   1:  PR[GP1:91,1] = PR[GP1:90,1] + 27.074;
   1:  PR[GP1:91,2] = PR[GP1:90,2] + -9.305;
   1:L PR[91] R[100]mm/sec CNT100;
   1:  PR[GP1:91,1] = PR[GP1:90,1] + 28.052;
   1:  PR[GP1:91,2] = PR[GP1:90,2] + -6.402;
   1:L PR[91] R[100]mm/sec CNT100;
   1:  PR[GP1:91,1] = PR[GP1:90,1] + 28.426;
   1:  PR[GP1:91,2] = PR[GP1:90,2] + -3.528;
   1:L PR[91] R[100]mm/sec CNT100;
   1:  PR[GP1:91,1] = PR[GP1:90,1] + 28.781;
   1:  PR[GP1:91,2] = PR[GP1:90,2] + -0.326;
   1:L PR[91] R[100]mm/sec CNT100;
   1:  PR[GP1:91,1] = PR[GP1:90,1] + 28.412;
   1:  PR[GP1:91,2] = PR[GP1:90,2] + 2.511;
   1:L PR[91] R[100]mm/sec CNT100;
   1:  PR[GP1:91,1] = PR[GP1:90,1] + 28.089;
   1:  PR[GP1:91,2] = PR[GP1:90,2] + 5.607;
   1:L PR[91] R[100]mm/sec CNT100;
   1:  PR[GP1:91,1] = PR[GP1:90,1] + 27.206;
   1:  PR[GP1:91,2] = PR[GP1:90,2] + 8.384;
   1:L PR[91] R[100]mm/sec CNT100;
   1:  PR[GP1:91,1] = PR[GP1:90,1] + 26.117;
   1:  PR[GP1:91,2] = PR[GP1:90,2] + 11.033;
   1:L PR[91] R[100]mm/sec CNT100;
   1:  PR[GP1:91,1] = PR[GP1:90,1] + 24.650;
   1:  PR[GP1:91,2] = PR[GP1:90,2] + 13.658;
   1:L PR[91] R[100]mm/sec CNT100;
   1:  PR[GP1:91,1] = PR[GP1:90,1] + 22.947;
   1:  PR[GP1:91,2] = PR[GP1:90,2] + 15.921;
   1:L PR[91] R[100]mm/sec CNT100;
   1:  PR[GP1:91,1] = PR[GP1:90,1] + 20.753;
   1:  PR[GP1:91,2] = PR[GP1:90,2] + 18.419;
   1:L PR[91] R[100]mm/sec CNT100;
   1:  PR[GP1:91,1] = PR[GP1:90,1] + 18.590;
   1:  PR[GP1:91,2] = PR[GP1:90,2] + 20.133;
   1:L PR[91] R[100]mm/sec CNT100;
   1:  PR[GP1:91,1] = PR[GP1:90,1] + 15.465;
   1:  PR[GP1:91,2] = PR[GP1:90,2] + 22.345;
   1:L PR[91] R[100]mm/sec CNT100;
   1:  PR[GP1:91,1] = PR[GP1:90,1] + 13.026;
   1:  PR[GP1:91,2] = PR[GP1:90,2] + 23.427;
   1:L PR[91] R[100]mm/sec CNT100;
   1:  PR[GP1:91,1] = PR[GP1:90,1] + 9.359;
   1:  PR[GP1:91,2] = PR[GP1:90,2] + 24.848;
   1:L PR[91] R[100]mm/sec CNT100;
   1:  PR[GP1:91,1] = PR[GP1:90,1] + 6.820;
   1:  PR[GP1:91,2] = PR[GP1:90,2] + 25.271;
   1:L PR[91] R[100]mm/sec CNT100;
   1:  PR[GP1:91,1] = PR[GP1:90,1] + 2.805;
   1:  PR[GP1:91,2] = PR[GP1:90,2] + 25.769;
   1:L PR[91] R[100]mm/sec CNT100;
   1:  PR[GP1:91,1] = PR[GP1:90,1] + 0.266;
   1:  PR[GP1:91,2] = PR[GP1:90,2] + 25.578;
   1:L PR[91] R[100]mm/sec CNT100;
   1:  PR[91] = PR[90];
   1:  PR[GP1:91,1] = PR[GP1:90,1] + -0.092;
   1:  PR[GP1:91,2] = PR[GP1:90,2] + 25.736;
   1:  PR[GP1:91,3] = PR[GP1:90,3] + 68.625;
   1:L PR[91] R[100]mm/sec CNT100;
   1:  PR[GP1:91,1] = PR[GP1:90,1] + -2.390;
   1:  PR[GP1:91,2] = PR[GP1:90,2] + 25.906;
   1:L PR[91] R[100]mm/sec CNT100;
   1:  PR[GP1:91,1] = PR[GP1:90,1] + -6.675;
   1:  PR[GP1:91,2] = PR[GP1:90,2] + 25.375;
   1:L PR[91] R[100]mm/sec CNT100;
   1:  PR[GP1:91,1] = PR[GP1:90,1] + -8.961;
   1:  PR[GP1:91,2] = PR[GP1:90,2] + 24.994;
   1:L PR[91] R[100]mm/sec CNT100;
   1:  PR[GP1:91,1] = PR[GP1:90,1] + -12.889;
   1:  PR[GP1:91,2] = PR[GP1:90,2] + 23.472;
   1:L PR[91] R[100]mm/sec CNT100;
   1:  PR[GP1:91,1] = PR[GP1:90,1] + -15.085;
   1:  PR[GP1:91,2] = PR[GP1:90,2] + 22.498;
   1:L PR[91] R[100]mm/sec CNT100;
   1:  PR[GP1:91,1] = PR[GP1:90,1] + -18.448;
   1:  PR[GP1:91,2] = PR[GP1:90,2] + 20.117;
   1:L PR[91] R[100]mm/sec CNT100;
   1:  PR[GP1:91,1] = PR[GP1:90,1] + -20.400;
   1:  PR[GP1:91,2] = PR[GP1:90,2] + 18.570;
   1:L PR[91] R[100]mm/sec CNT100;
   1:  PR[GP1:91,1] = PR[GP1:90,1] + -22.619;
   1:  PR[GP1:91,2] = PR[GP1:90,2] + 16.084;
   1:L PR[91] R[100]mm/sec CNT100;
   1:  PR[GP1:91,1] = PR[GP1:90,1] + -24.160;
   1:  PR[GP1:91,2] = PR[GP1:90,2] + 14.037;
   1:L PR[91] R[100]mm/sec CNT100;
   1:  PR[GP1:91,1] = PR[GP1:90,1] + -25.748;
   1:  PR[GP1:91,2] = PR[GP1:90,2] + 11.314;
   1:L PR[91] R[100]mm/sec CNT100;
   1:  PR[GP1:91,1] = PR[GP1:90,1] + -26.729;
   1:  PR[GP1:91,2] = PR[GP1:90,2] + 8.924;
   1:L PR[91] R[100]mm/sec CNT100;
   1:  PR[GP1:91,1] = PR[GP1:90,1] + -27.794;
   1:  PR[GP1:91,2] = PR[GP1:90,2] + 5.767;
   1:L PR[91] R[100]mm/sec CNT100;
   1:  PR[GP1:91,1] = PR[GP1:90,1] + -28.130;
   1:  PR[GP1:91,2] = PR[GP1:90,2] + 3.188;
   1:L PR[91] R[100]mm/sec CNT100;
   1:  PR[GP1:91,1] = PR[GP1:90,1] + -28.516;
   1:  PR[GP1:91,2] = PR[GP1:90,2] + -0.298;
   1:L PR[91] R[100]mm/sec CNT100;
   1:  PR[GP1:91,1] = PR[GP1:90,1] + -28.184;
   1:  PR[GP1:91,2] = PR[GP1:90,2] + -2.847;
   1:L PR[91] R[100]mm/sec CNT100;
   1:  PR[GP1:91,1] = PR[GP1:90,1] + -27.833;
   1:  PR[GP1:91,2] = PR[GP1:90,2] + -6.208;
   1:L PR[91] R[100]mm/sec CNT100;
   1:  PR[GP1:91,1] = PR[GP1:90,1] + -26.872;
   1:  PR[GP1:91,2] = PR[GP1:90,2] + -9.231;
   1:L PR[91] R[100]mm/sec CNT100;
   1:  PR[GP1:91,1] = PR[GP1:90,1] + -25.890;
   1:  PR[GP1:91,2] = PR[GP1:90,2] + -11.618;
   1:L PR[91] R[100]mm/sec CNT100;
   1:  PR[GP1:91,1] = PR[GP1:90,1] + -24.299;
   1:  PR[GP1:91,2] = PR[GP1:90,2] + -14.466;
   1:L PR[91] R[100]mm/sec CNT100;
   1:  PR[GP1:91,1] = PR[GP1:90,1] + -22.763;
   1:  PR[GP1:91,2] = PR[GP1:90,2] + -16.503;
   1:L PR[91] R[100]mm/sec CNT100;
   1:  PR[GP1:91,1] = PR[GP1:90,1] + -20.390;
   1:  PR[GP1:91,2] = PR[GP1:90,2] + -19.204;
   1:L PR[91] R[100]mm/sec CNT100;
   1:  PR[GP1:91,1] = PR[GP1:90,1] + -16.718;
   1:  PR[GP1:91,2] = PR[GP1:90,2] + -22.122;
   1:L PR[91] R[100]mm/sec CNT100;
   1:  PR[GP1:91,1] = PR[GP1:90,1] + -14.983;
   1:  PR[GP1:91,2] = PR[GP1:90,2] + -23.178;
   1:L PR[91] R[100]mm/sec CNT100;
   1:  PR[GP1:91,1] = PR[GP1:90,1] + -12.771;
   1:  PR[GP1:91,2] = PR[GP1:90,2] + -24.157;
   1:L PR[91] R[100]mm/sec CNT100;
   1:  PR[GP1:91,1] = PR[GP1:90,1] + -8.827;
   1:  PR[GP1:91,2] = PR[GP1:90,2] + -25.648;
   1:L PR[91] R[100]mm/sec CNT100;
   1:  PR[GP1:91,1] = PR[GP1:90,1] + -6.599;
   1:  PR[GP1:91,2] = PR[GP1:90,2] + -26.016;
   1:L PR[91] R[100]mm/sec CNT100;
   1:  PR[GP1:91,1] = PR[GP1:90,1] + -2.291;
   1:  PR[GP1:91,2] = PR[GP1:90,2] + -26.524;
   1:L PR[91] R[100]mm/sec CNT100;
   1:  PR[GP1:91,1] = PR[GP1:90,1] + -0.100;
   1:  PR[GP1:91,2] = PR[GP1:90,2] + -26.354;
   1:L PR[91] R[100]mm/sec CNT100;
   1:  PR[GP1:91,1] = PR[GP1:90,1] + 0.256;
   1:L PR[91] R[100]mm/sec CNT100;
   1:  PR[GP1:91,1] = PR[GP1:90,1] + 2.490;
   1:  PR[GP1:91,2] = PR[GP1:90,2] + -26.527;
   1:L PR[91] R[100]mm/sec CNT100;
   1:  PR[GP1:91,1] = PR[GP1:90,1] + 4.700;
   1:  PR[GP1:91,2] = PR[GP1:90,2] + -26.395;
   1:L PR[91] R[100]mm/sec CNT100;
   1:  PR[GP1:91,1] = PR[GP1:90,1] + 7.039;
   1:  PR[GP1:91,2] = PR[GP1:90,2] + -26.007;
   1:L PR[91] R[100]mm/sec CNT100;
   1:  PR[GP1:91,1] = PR[GP1:90,1] + 9.138;
   1:  PR[GP1:91,2] = PR[GP1:90,2] + -25.611;
   1:L PR[91] R[100]mm/sec CNT100;
   1:  PR[GP1:91,1] = PR[GP1:90,1] + 13.058;
   1:  PR[GP1:91,2] = PR[GP1:90,2] + -24.087;
   1:L PR[91] R[100]mm/sec CNT100;
   1:  PR[GP1:91,1] = PR[GP1:90,1] + 15.230;
   1:  PR[GP1:91,2] = PR[GP1:90,2] + -23.127;
   1:L PR[91] R[100]mm/sec CNT100;
   1:  PR[GP1:91,1] = PR[GP1:90,1] + 18.598;
   1:  PR[GP1:91,2] = PR[GP1:90,2] + -20.745;
   1:L PR[91] R[100]mm/sec CNT100;
   1:  PR[GP1:91,1] = PR[GP1:90,1] + 20.553;
   1:  PR[GP1:91,2] = PR[GP1:90,2] + -19.198;
   1:L PR[91] R[100]mm/sec CNT100;
   1:  PR[GP1:91,1] = PR[GP1:90,1] + 22.771;
   1:  PR[GP1:91,2] = PR[GP1:90,2] + -16.712;
   1:L PR[91] R[100]mm/sec CNT100;
   1:  PR[GP1:91,1] = PR[GP1:90,1] + 24.315;
   1:  PR[GP1:91,2] = PR[GP1:90,2] + -14.663;
   1:L PR[91] R[100]mm/sec CNT100;
   1:  PR[GP1:91,1] = PR[GP1:90,1] + 25.903;
   1:  PR[GP1:91,2] = PR[GP1:90,2] + -11.940;
   1:L PR[91] R[100]mm/sec CNT100;
   1:  PR[GP1:91,1] = PR[GP1:90,1] + 26.886;
   1:  PR[GP1:91,2] = PR[GP1:90,2] + -9.552;
   1:L PR[91] R[100]mm/sec CNT100;
   1:  PR[GP1:91,1] = PR[GP1:90,1] + 27.950;
   1:  PR[GP1:91,2] = PR[GP1:90,2] + -6.395;
   1:L PR[91] R[100]mm/sec CNT100;
   1:  PR[GP1:91,1] = PR[GP1:90,1] + 28.287;
   1:  PR[GP1:91,2] = PR[GP1:90,2] + -3.812;
   1:L PR[91] R[100]mm/sec CNT100;
   1:  PR[GP1:91,1] = PR[GP1:90,1] + 28.673;
   1:  PR[GP1:91,2] = PR[GP1:90,2] + -0.326;
   1:L PR[91] R[100]mm/sec CNT100;
   1:  PR[GP1:91,1] = PR[GP1:90,1] + 28.341;
   1:  PR[GP1:91,2] = PR[GP1:90,2] + 2.223;
   1:L PR[91] R[100]mm/sec CNT100;
   1:  PR[GP1:91,1] = PR[GP1:90,1] + 27.991;
   1:  PR[GP1:91,2] = PR[GP1:90,2] + 5.583;
   1:L PR[91] R[100]mm/sec CNT100;
   1:  PR[GP1:91,1] = PR[GP1:90,1] + 27.030;
   1:  PR[GP1:91,2] = PR[GP1:90,2] + 8.605;
   1:L PR[91] R[100]mm/sec CNT100;
   1:  PR[GP1:91,1] = PR[GP1:90,1] + 26.050;
   1:  PR[GP1:91,2] = PR[GP1:90,2] + 10.988;
   1:L PR[91] R[100]mm/sec CNT100;
   1:  PR[GP1:91,1] = PR[GP1:90,1] + 24.458;
   1:  PR[GP1:91,2] = PR[GP1:90,2] + 13.836;
   1:L PR[91] R[100]mm/sec CNT100;
   1:  PR[GP1:91,1] = PR[GP1:90,1] + 22.926;
   1:  PR[GP1:91,2] = PR[GP1:90,2] + 15.873;
   1:L PR[91] R[100]mm/sec CNT100;
   1:  PR[GP1:91,1] = PR[GP1:90,1] + 20.554;
   1:  PR[GP1:91,2] = PR[GP1:90,2] + 18.573;
   1:L PR[91] R[100]mm/sec CNT100;
   1:  PR[GP1:91,1] = PR[GP1:90,1] + 18.605;
   1:  PR[GP1:91,2] = PR[GP1:90,2] + 20.117;
   1:L PR[91] R[100]mm/sec CNT100;
   1:  PR[GP1:91,1] = PR[GP1:90,1] + 15.243;
   1:  PR[GP1:91,2] = PR[GP1:90,2] + 22.498;
   1:L PR[91] R[100]mm/sec CNT100;
   1:  PR[GP1:91,1] = PR[GP1:90,1] + 13.047;
   1:  PR[GP1:91,2] = PR[GP1:90,2] + 23.472;
   1:L PR[91] R[100]mm/sec CNT100;
   1:  PR[GP1:91,1] = PR[GP1:90,1] + 9.117;
   1:  PR[GP1:91,2] = PR[GP1:90,2] + 24.994;
   1:L PR[91] R[100]mm/sec CNT100;
   1:  PR[GP1:91,1] = PR[GP1:90,1] + 6.832;
   1:  PR[GP1:91,2] = PR[GP1:90,2] + 25.375;
   1:L PR[91] R[100]mm/sec CNT100;
   1:  PR[GP1:91,1] = PR[GP1:90,1] + 2.546;
   1:  PR[GP1:91,2] = PR[GP1:90,2] + 25.906;
   1:L PR[91] R[100]mm/sec CNT100;
   1:  PR[GP1:91,1] = PR[GP1:90,1] + 0.252;
   1:  PR[GP1:91,2] = PR[GP1:90,2] + 25.736;
   1:L PR[91] R[100]mm/sec CNT100;
   1:  PR[91] = PR[90];
   1:  PR[GP1:91,1] = PR[GP1:90,1] + -0.083;
   1:  PR[GP1:91,2] = PR[GP1:90,2] + 25.892;
   1:  PR[GP1:91,3] = PR[GP1:90,3] + 69.235;
   1:L PR[91] R[100]mm/sec CNT100;
   1:  PR[GP1:91,1] = PR[GP1:90,1] + -2.132;
   1:  PR[GP1:91,2] = PR[GP1:90,2] + 26.044;
   1:L PR[91] R[100]mm/sec CNT100;
   1:  PR[GP1:91,1] = PR[GP1:90,1] + -6.687;
   1:  PR[GP1:91,2] = PR[GP1:90,2] + 25.479;
   1:L PR[91] R[100]mm/sec CNT100;
   1:  PR[GP1:91,1] = PR[GP1:90,1] + -8.719;
   1:  PR[GP1:91,2] = PR[GP1:90,2] + 25.141;
   1:L PR[91] R[100]mm/sec CNT100;
   1:  PR[GP1:91,1] = PR[GP1:90,1] + -12.910;
   1:  PR[GP1:91,2] = PR[GP1:90,2] + 23.517;
   1:L PR[91] R[100]mm/sec CNT100;
   1:  PR[GP1:91,1] = PR[GP1:90,1] + -14.863;
   1:  PR[GP1:91,2] = PR[GP1:90,2] + 22.650;
   1:L PR[91] R[100]mm/sec CNT100;
   1:  PR[GP1:91,1] = PR[GP1:90,1] + -18.463;
   1:  PR[GP1:91,2] = PR[GP1:90,2] + 20.101;
   1:L PR[91] R[100]mm/sec CNT100;
   1:  PR[GP1:91,1] = PR[GP1:90,1] + -20.201;
   1:  PR[GP1:91,2] = PR[GP1:90,2] + 18.724;
   1:L PR[91] R[100]mm/sec CNT100;
   1:  PR[GP1:91,1] = PR[GP1:90,1] + -22.586;
   1:  PR[GP1:91,2] = PR[GP1:90,2] + 16.051;
   1:L PR[91] R[100]mm/sec CNT100;
   1:  PR[GP1:91,1] = PR[GP1:90,1] + -23.957;
   1:  PR[GP1:91,2] = PR[GP1:90,2] + 14.230;
   1:L PR[91] R[100]mm/sec CNT100;
   1:  PR[GP1:91,1] = PR[GP1:90,1] + -25.670;
   1:  PR[GP1:91,2] = PR[GP1:90,2] + 11.294;
   1:L PR[91] R[100]mm/sec CNT100;
   1:  PR[GP1:91,1] = PR[GP1:90,1] + -26.542;
   1:  PR[GP1:91,2] = PR[GP1:90,2] + 9.171;
   1:L PR[91] R[100]mm/sec CNT100;
   1:  PR[GP1:91,1] = PR[GP1:90,1] + -27.692;
   1:  PR[GP1:91,2] = PR[GP1:90,2] + 5.760;
   1:L PR[91] R[100]mm/sec CNT100;
   1:  PR[GP1:91,1] = PR[GP1:90,1] + -27.990;
   1:  PR[GP1:91,2] = PR[GP1:90,2] + 3.472;
   1:L PR[91] R[100]mm/sec CNT100;
   1:  PR[GP1:91,1] = PR[GP1:90,1] + -28.408;
   1:  PR[GP1:91,2] = PR[GP1:90,2] + -0.298;
   1:L PR[91] R[100]mm/sec CNT100;
   1:  PR[GP1:91,1] = PR[GP1:90,1] + -28.113;
   1:  PR[GP1:91,2] = PR[GP1:90,2] + -2.558;
   1:L PR[91] R[100]mm/sec CNT100;
   1:  PR[GP1:91,1] = PR[GP1:90,1] + -27.735;
   1:  PR[GP1:91,2] = PR[GP1:90,2] + -6.185;
   1:L PR[91] R[100]mm/sec CNT100;
   1:  PR[GP1:91,1] = PR[GP1:90,1] + -26.696;
   1:  PR[GP1:91,2] = PR[GP1:90,2] + -9.452;
   1:L PR[91] R[100]mm/sec CNT100;
   1:  PR[GP1:91,1] = PR[GP1:90,1] + -25.824;
   1:  PR[GP1:91,2] = PR[GP1:90,2] + -11.573;
   1:L PR[91] R[100]mm/sec CNT100;
   1:  PR[GP1:91,1] = PR[GP1:90,1] + -24.108;
   1:  PR[GP1:91,2] = PR[GP1:90,2] + -14.643;
   1:L PR[91] R[100]mm/sec CNT100;
   1:  PR[GP1:91,1] = PR[GP1:90,1] + -22.742;
   1:  PR[GP1:91,2] = PR[GP1:90,2] + -16.454;
   1:L PR[91] R[100]mm/sec CNT100;
   1:  PR[GP1:91,1] = PR[GP1:90,1] + -20.191;
   1:  PR[GP1:91,2] = PR[GP1:90,2] + -19.357;
   1:L PR[91] R[100]mm/sec CNT100;
   1:  PR[GP1:91,1] = PR[GP1:90,1] + -16.615;
   1:  PR[GP1:91,2] = PR[GP1:90,2] + -22.201;
   1:L PR[91] R[100]mm/sec CNT100;
   1:  PR[GP1:91,1] = PR[GP1:90,1] + -14.753;
   1:  PR[GP1:91,2] = PR[GP1:90,2] + -23.335;
   1:L PR[91] R[100]mm/sec CNT100;
   1:  PR[GP1:91,1] = PR[GP1:90,1] + -12.786;
   1:  PR[GP1:91,2] = PR[GP1:90,2] + -24.205;
   1:L PR[91] R[100]mm/sec CNT100;
   1:  PR[GP1:91,1] = PR[GP1:90,1] + -8.578;
   1:  PR[GP1:91,2] = PR[GP1:90,2] + -25.796;
   1:L PR[91] R[100]mm/sec CNT100;
   1:  PR[GP1:91,1] = PR[GP1:90,1] + -6.608;
   1:  PR[GP1:91,2] = PR[GP1:90,2] + -26.121;
   1:L PR[91] R[100]mm/sec CNT100;
   1:  PR[GP1:91,1] = PR[GP1:90,1] + -2.029;
   1:  PR[GP1:91,2] = PR[GP1:90,2] + -26.661;
   1:L PR[91] R[100]mm/sec CNT100;
   1:  PR[GP1:91,1] = PR[GP1:90,1] + -0.087;
   1:  PR[GP1:91,2] = PR[GP1:90,2] + -26.510;
   1:L PR[91] R[100]mm/sec CNT100;
   1:  PR[GP1:91,1] = PR[GP1:90,1] + 0.244;
   1:L PR[91] R[100]mm/sec CNT100;
   1:  PR[GP1:91,1] = PR[GP1:90,1] + 2.228;
   1:  PR[GP1:91,2] = PR[GP1:90,2] + -26.664;
   1:L PR[91] R[100]mm/sec CNT100;
   1:  PR[GP1:91,1] = PR[GP1:90,1] + 4.582;
   1:  PR[GP1:91,2] = PR[GP1:90,2] + -26.524;
   1:L PR[91] R[100]mm/sec CNT100;
   1:  PR[GP1:91,1] = PR[GP1:90,1] + 6.658;
   1:  PR[GP1:91,2] = PR[GP1:90,2] + -26.179;
   1:L PR[91] R[100]mm/sec CNT100;
   1:  PR[GP1:91,1] = PR[GP1:90,1] + 8.901;
   1:  PR[GP1:91,2] = PR[GP1:90,2] + -25.756;
   1:L PR[91] R[100]mm/sec CNT100;
   1:  PR[GP1:91,1] = PR[GP1:90,1] + 13.082;
   1:  PR[GP1:91,2] = PR[GP1:90,2] + -24.130;
   1:L PR[91] R[100]mm/sec CNT100;
   1:  PR[GP1:91,1] = PR[GP1:90,1] + 15.008;
   1:  PR[GP1:91,2] = PR[GP1:90,2] + -23.279;
   1:L PR[91] R[100]mm/sec CNT100;
   1:  PR[GP1:91,1] = PR[GP1:90,1] + 18.614;
   1:  PR[GP1:91,2] = PR[GP1:90,2] + -20.729;
   1:L PR[91] R[100]mm/sec CNT100;
   1:  PR[GP1:91,1] = PR[GP1:90,1] + 20.355;
   1:  PR[GP1:91,2] = PR[GP1:90,2] + -19.352;
   1:L PR[91] R[100]mm/sec CNT100;
   1:  PR[GP1:91,1] = PR[GP1:90,1] + 22.740;
   1:  PR[GP1:91,2] = PR[GP1:90,2] + -16.679;
   1:L PR[91] R[100]mm/sec CNT100;
   1:  PR[GP1:91,1] = PR[GP1:90,1] + 24.113;
   1:  PR[GP1:91,2] = PR[GP1:90,2] + -14.856;
   1:L PR[91] R[100]mm/sec CNT100;
   1:  PR[GP1:91,1] = PR[GP1:90,1] + 25.825;
   1:  PR[GP1:91,2] = PR[GP1:90,2] + -11.919;
   1:L PR[91] R[100]mm/sec CNT100;
   1:  PR[GP1:91,1] = PR[GP1:90,1] + 26.699;
   1:  PR[GP1:91,2] = PR[GP1:90,2] + -9.798;
   1:L PR[91] R[100]mm/sec CNT100;
   1:  PR[GP1:91,1] = PR[GP1:90,1] + 27.848;
   1:  PR[GP1:91,2] = PR[GP1:90,2] + -6.388;
   1:L PR[91] R[100]mm/sec CNT100;
   1:  PR[GP1:91,1] = PR[GP1:90,1] + 28.147;
   1:  PR[GP1:91,2] = PR[GP1:90,2] + -4.096;
   1:L PR[91] R[100]mm/sec CNT100;
   1:  PR[GP1:91,1] = PR[GP1:90,1] + 28.564;
   1:  PR[GP1:91,2] = PR[GP1:90,2] + -0.326;
   1:L PR[91] R[100]mm/sec CNT100;
   1:  PR[GP1:91,1] = PR[GP1:90,1] + 28.270;
   1:  PR[GP1:91,2] = PR[GP1:90,2] + 1.934;
   1:L PR[91] R[100]mm/sec CNT100;
   1:  PR[GP1:91,1] = PR[GP1:90,1] + 27.892;
   1:  PR[GP1:91,2] = PR[GP1:90,2] + 5.560;
   1:L PR[91] R[100]mm/sec CNT100;
   1:  PR[GP1:91,1] = PR[GP1:90,1] + 26.853;
   1:  PR[GP1:91,2] = PR[GP1:90,2] + 8.827;
   1:L PR[91] R[100]mm/sec CNT100;
   1:  PR[GP1:91,1] = PR[GP1:90,1] + 25.983;
   1:  PR[GP1:91,2] = PR[GP1:90,2] + 10.943;
   1:L PR[91] R[100]mm/sec CNT100;
   1:  PR[GP1:91,1] = PR[GP1:90,1] + 24.267;
   1:  PR[GP1:91,2] = PR[GP1:90,2] + 14.014;
   1:L PR[91] R[100]mm/sec CNT100;
   1:  PR[GP1:91,1] = PR[GP1:90,1] + 22.904;
   1:  PR[GP1:91,2] = PR[GP1:90,2] + 15.825;
   1:L PR[91] R[100]mm/sec CNT100;
   1:  PR[GP1:91,1] = PR[GP1:90,1] + 20.355;
   1:  PR[GP1:91,2] = PR[GP1:90,2] + 18.727;
   1:L PR[91] R[100]mm/sec CNT100;
   1:  PR[GP1:91,1] = PR[GP1:90,1] + 18.621;
   1:  PR[GP1:91,2] = PR[GP1:90,2] + 20.101;
   1:L PR[91] R[100]mm/sec CNT100;
   1:  PR[GP1:91,1] = PR[GP1:90,1] + 15.020;
   1:  PR[GP1:91,2] = PR[GP1:90,2] + 22.650;
   1:L PR[91] R[100]mm/sec CNT100;
   1:  PR[GP1:91,1] = PR[GP1:90,1] + 13.068;
   1:  PR[GP1:91,2] = PR[GP1:90,2] + 23.516;
   1:L PR[91] R[100]mm/sec CNT100;
   1:  PR[GP1:91,1] = PR[GP1:90,1] + 8.876;
   1:  PR[GP1:91,2] = PR[GP1:90,2] + 25.141;
   1:L PR[91] R[100]mm/sec CNT100;
   1:  PR[GP1:91,1] = PR[GP1:90,1] + 6.844;
   1:  PR[GP1:91,2] = PR[GP1:90,2] + 25.480;
   1:L PR[91] R[100]mm/sec CNT100;
   1:  PR[GP1:91,1] = PR[GP1:90,1] + 2.288;
   1:  PR[GP1:91,2] = PR[GP1:90,2] + 26.044;
   1:L PR[91] R[100]mm/sec CNT100;
   1:  PR[GP1:91,1] = PR[GP1:90,1] + 0.239;
   1:  PR[GP1:91,2] = PR[GP1:90,2] + 25.892;
   1:L PR[91] R[100]mm/sec CNT100;
   1:  PR[91] = PR[90];
   1:  PR[GP1:91,1] = PR[GP1:90,1] + -0.070;
   1:  PR[GP1:91,2] = PR[GP1:90,2] + 26.047;
   1:  PR[GP1:91,3] = PR[GP1:90,3] + 69.845;
   1:L PR[91] R[100]mm/sec CNT100;
   1:  PR[GP1:91,1] = PR[GP1:90,1] + -1.874;
   1:  PR[GP1:91,2] = PR[GP1:90,2] + 26.181;
   1:L PR[91] R[100]mm/sec CNT100;
   1:  PR[GP1:91,1] = PR[GP1:90,1] + -6.699;
   1:  PR[GP1:91,2] = PR[GP1:90,2] + 25.584;
   1:L PR[91] R[100]mm/sec CNT100;
   1:  PR[GP1:91,1] = PR[GP1:90,1] + -8.478;
   1:  PR[GP1:91,2] = PR[GP1:90,2] + 25.287;
   1:L PR[91] R[100]mm/sec CNT100;
   1:  PR[GP1:91,1] = PR[GP1:90,1] + -12.931;
   1:  PR[GP1:91,2] = PR[GP1:90,2] + 23.561;
   1:L PR[91] R[100]mm/sec CNT100;
   1:  PR[GP1:91,1] = PR[GP1:90,1] + -14.641;
   1:  PR[GP1:91,2] = PR[GP1:90,2] + 22.803;
   1:L PR[91] R[100]mm/sec CNT100;
   1:  PR[GP1:91,1] = PR[GP1:90,1] + -18.478;
   1:  PR[GP1:91,2] = PR[GP1:90,2] + 20.085;
   1:L PR[91] R[100]mm/sec CNT100;
   1:  PR[GP1:91,1] = PR[GP1:90,1] + -20.003;
   1:  PR[GP1:91,2] = PR[GP1:90,2] + 18.878;
   1:L PR[91] R[100]mm/sec CNT100;
   1:  PR[GP1:91,1] = PR[GP1:90,1] + -22.554;
   1:  PR[GP1:91,2] = PR[GP1:90,2] + 16.018;
   1:L PR[91] R[100]mm/sec CNT100;
   1:  PR[GP1:91,1] = PR[GP1:90,1] + -23.755;
   1:  PR[GP1:91,2] = PR[GP1:90,2] + 14.424;
   1:L PR[91] R[100]mm/sec CNT100;
   1:  PR[GP1:91,1] = PR[GP1:90,1] + -25.592;
   1:  PR[GP1:91,2] = PR[GP1:90,2] + 11.274;
   1:L PR[91] R[100]mm/sec CNT100;
   1:  PR[GP1:91,1] = PR[GP1:90,1] + -26.354;
   1:  PR[GP1:91,2] = PR[GP1:90,2] + 9.418;
   1:L PR[91] R[100]mm/sec CNT100;
   1:  PR[GP1:91,1] = PR[GP1:90,1] + -27.590;
   1:  PR[GP1:91,2] = PR[GP1:90,2] + 5.753;
   1:L PR[91] R[100]mm/sec CNT100;
   1:  PR[GP1:91,1] = PR[GP1:90,1] + -27.850;
   1:  PR[GP1:91,2] = PR[GP1:90,2] + 3.756;
   1:L PR[91] R[100]mm/sec CNT100;
   1:  PR[GP1:91,1] = PR[GP1:90,1] + -28.299;
   1:  PR[GP1:91,2] = PR[GP1:90,2] + -0.298;
   1:L PR[91] R[100]mm/sec CNT100;
   1:  PR[GP1:91,1] = PR[GP1:90,1] + -28.042;
   1:  PR[GP1:91,2] = PR[GP1:90,2] + -2.270;
   1:L PR[91] R[100]mm/sec CNT100;
   1:  PR[GP1:91,1] = PR[GP1:90,1] + -27.636;
   1:  PR[GP1:91,2] = PR[GP1:90,2] + -6.162;
   1:L PR[91] R[100]mm/sec CNT100;
   1:  PR[GP1:91,1] = PR[GP1:90,1] + -26.519;
   1:  PR[GP1:91,2] = PR[GP1:90,2] + -9.673;
   1:L PR[91] R[100]mm/sec CNT100;
   1:  PR[GP1:91,1] = PR[GP1:90,1] + -25.757;
   1:  PR[GP1:91,2] = PR[GP1:90,2] + -11.527;
   1:L PR[91] R[100]mm/sec CNT100;
   1:  PR[GP1:91,1] = PR[GP1:90,1] + -23.916;
   1:  PR[GP1:91,2] = PR[GP1:90,2] + -14.821;
   1:L PR[91] R[100]mm/sec CNT100;
   1:  PR[GP1:91,1] = PR[GP1:90,1] + -22.722;
   1:  PR[GP1:91,2] = PR[GP1:90,2] + -16.406;
   1:L PR[91] R[100]mm/sec CNT100;
   1:  PR[GP1:91,1] = PR[GP1:90,1] + -19.993;
   1:  PR[GP1:91,2] = PR[GP1:90,2] + -19.511;
   1:L PR[91] R[100]mm/sec CNT100;
   1:  PR[GP1:91,1] = PR[GP1:90,1] + -16.512;
   1:  PR[GP1:91,2] = PR[GP1:90,2] + -22.280;
   1:L PR[91] R[100]mm/sec CNT100;
   1:  PR[GP1:91,1] = PR[GP1:90,1] + -14.522;
   1:  PR[GP1:91,2] = PR[GP1:90,2] + -23.491;
   1:L PR[91] R[100]mm/sec CNT100;
   1:  PR[GP1:91,1] = PR[GP1:90,1] + -12.801;
   1:  PR[GP1:91,2] = PR[GP1:90,2] + -24.253;
   1:L PR[91] R[100]mm/sec CNT100;
   1:  PR[GP1:91,1] = PR[GP1:90,1] + -8.330;
   1:  PR[GP1:91,2] = PR[GP1:90,2] + -25.943;
   1:L PR[91] R[100]mm/sec CNT100;
   1:  PR[GP1:91,1] = PR[GP1:90,1] + -6.618;
   1:  PR[GP1:91,2] = PR[GP1:90,2] + -26.226;
   1:L PR[91] R[100]mm/sec CNT100;
   1:  PR[GP1:91,1] = PR[GP1:90,1] + -1.767;
   1:  PR[GP1:91,2] = PR[GP1:90,2] + -26.798;
   1:L PR[91] R[100]mm/sec CNT100;
   1:  PR[GP1:91,1] = PR[GP1:90,1] + -0.074;
   1:  PR[GP1:91,2] = PR[GP1:90,2] + -26.667;
   1:L PR[91] R[100]mm/sec CNT100;
   1:  PR[GP1:91,1] = PR[GP1:90,1] + 0.231;
   1:L PR[91] R[100]mm/sec CNT100;
   1:  PR[GP1:91,1] = PR[GP1:90,1] + 1.966;
   1:  PR[GP1:91,2] = PR[GP1:90,2] + -26.802;
   1:L PR[91] R[100]mm/sec CNT100;
   1:  PR[GP1:91,1] = PR[GP1:90,1] + 4.464;
   1:  PR[GP1:91,2] = PR[GP1:90,2] + -26.652;
   1:L PR[91] R[100]mm/sec CNT100;
   1:  PR[GP1:91,1] = PR[GP1:90,1] + 6.277;
   1:  PR[GP1:91,2] = PR[GP1:90,2] + -26.352;
   1:L PR[91] R[100]mm/sec CNT100;
   1:  PR[GP1:91,1] = PR[GP1:90,1] + 8.663;
   1:  PR[GP1:91,2] = PR[GP1:90,2] + -25.901;
   1:L PR[91] R[100]mm/sec CNT100;
   1:  PR[GP1:91,1] = PR[GP1:90,1] + 13.105;
   1:  PR[GP1:91,2] = PR[GP1:90,2] + -24.174;
   1:L PR[91] R[100]mm/sec CNT100;
   1:  PR[GP1:91,1] = PR[GP1:90,1] + 14.786;
   1:  PR[GP1:91,2] = PR[GP1:90,2] + -23.431;
   1:L PR[91] R[100]mm/sec CNT100;
   1:  PR[GP1:91,1] = PR[GP1:90,1] + 18.630;
   1:  PR[GP1:91,2] = PR[GP1:90,2] + -20.712;
   1:L PR[91] R[100]mm/sec CNT100;
   1:  PR[GP1:91,1] = PR[GP1:90,1] + 20.156;
   1:  PR[GP1:91,2] = PR[GP1:90,2] + -19.505;
   1:L PR[91] R[100]mm/sec CNT100;
   1:  PR[GP1:91,1] = PR[GP1:90,1] + 22.708;
   1:  PR[GP1:91,2] = PR[GP1:90,2] + -16.645;
   1:L PR[91] R[100]mm/sec CNT100;
   1:  PR[GP1:91,1] = PR[GP1:90,1] + 23.910;
   1:  PR[GP1:91,2] = PR[GP1:90,2] + -15.049;
   1:L PR[91] R[100]mm/sec CNT100;
   1:  PR[GP1:91,1] = PR[GP1:90,1] + 25.748;
   1:  PR[GP1:91,2] = PR[GP1:90,2] + -11.899;
   1:L PR[91] R[100]mm/sec CNT100;
   1:  PR[GP1:91,1] = PR[GP1:90,1] + 26.511;
   1:  PR[GP1:91,2] = PR[GP1:90,2] + -10.044;
   1:L PR[91] R[100]mm/sec CNT100;
   1:  PR[GP1:91,1] = PR[GP1:90,1] + 27.746;
   1:  PR[GP1:91,2] = PR[GP1:90,2] + -6.381;
   1:L PR[91] R[100]mm/sec CNT100;
   1:  PR[GP1:91,1] = PR[GP1:90,1] + 28.007;
   1:  PR[GP1:91,2] = PR[GP1:90,2] + -4.380;
   1:L PR[91] R[100]mm/sec CNT100;
   1:  PR[GP1:91,1] = PR[GP1:90,1] + 28.456;
   1:  PR[GP1:91,2] = PR[GP1:90,2] + -0.326;
   1:L PR[91] R[100]mm/sec CNT100;
   1:  PR[GP1:91,1] = PR[GP1:90,1] + 28.199;
   1:  PR[GP1:91,2] = PR[GP1:90,2] + 1.646;
   1:L PR[91] R[100]mm/sec CNT100;
   1:  PR[GP1:91,1] = PR[GP1:90,1] + 27.794;
   1:  PR[GP1:91,2] = PR[GP1:90,2] + 5.537;
   1:L PR[91] R[100]mm/sec CNT100;
   1:  PR[GP1:91,1] = PR[GP1:90,1] + 26.677;
   1:  PR[GP1:91,2] = PR[GP1:90,2] + 9.048;
   1:L PR[91] R[100]mm/sec CNT100;
   1:  PR[GP1:91,1] = PR[GP1:90,1] + 25.916;
   1:  PR[GP1:91,2] = PR[GP1:90,2] + 10.898;
   1:L PR[91] R[100]mm/sec CNT100;
   1:  PR[GP1:91,1] = PR[GP1:90,1] + 24.076;
   1:  PR[GP1:91,2] = PR[GP1:90,2] + 14.192;
   1:L PR[91] R[100]mm/sec CNT100;
   1:  PR[GP1:91,1] = PR[GP1:90,1] + 22.883;
   1:  PR[GP1:91,2] = PR[GP1:90,2] + 15.777;
   1:L PR[91] R[100]mm/sec CNT100;
   1:  PR[GP1:91,1] = PR[GP1:90,1] + 20.156;
   1:  PR[GP1:91,2] = PR[GP1:90,2] + 18.881;
   1:L PR[91] R[100]mm/sec CNT100;
   1:  PR[GP1:91,1] = PR[GP1:90,1] + 18.636;
   1:  PR[GP1:91,2] = PR[GP1:90,2] + 20.085;
   1:L PR[91] R[100]mm/sec CNT100;
   1:  PR[GP1:91,1] = PR[GP1:90,1] + 14.798;
   1:  PR[GP1:91,2] = PR[GP1:90,2] + 22.803;
   1:L PR[91] R[100]mm/sec CNT100;
   1:  PR[GP1:91,1] = PR[GP1:90,1] + 13.088;
   1:  PR[GP1:91,2] = PR[GP1:90,2] + 23.561;
   1:L PR[91] R[100]mm/sec CNT100;
   1:  PR[GP1:91,1] = PR[GP1:90,1] + 8.634;
   1:  PR[GP1:91,2] = PR[GP1:90,2] + 25.287;
   1:L PR[91] R[100]mm/sec CNT100;
   1:  PR[GP1:91,1] = PR[GP1:90,1] + 6.856;
   1:  PR[GP1:91,2] = PR[GP1:90,2] + 25.584;
   1:L PR[91] R[100]mm/sec CNT100;
   1:  PR[GP1:91,1] = PR[GP1:90,1] + 2.030;
   1:  PR[GP1:91,2] = PR[GP1:90,2] + 26.181;
   1:L PR[91] R[100]mm/sec CNT100;
   1:  PR[GP1:91,1] = PR[GP1:90,1] + 0.227;
   1:  PR[GP1:91,2] = PR[GP1:90,2] + 26.047;
   1:L PR[91] R[100]mm/sec CNT100;
   1:  PR[91] = PR[90];
   1:  PR[GP1:91,1] = PR[GP1:90,1] + -0.058;
   1:  PR[GP1:91,2] = PR[GP1:90,2] + 26.203;
   1:  PR[GP1:91,3] = PR[GP1:90,3] + 70.455;
   1:L PR[91] R[100]mm/sec CNT100;
   1:  PR[GP1:91,1] = PR[GP1:90,1] + -1.617;
   1:  PR[GP1:91,2] = PR[GP1:90,2] + 26.319;
   1:L PR[91] R[100]mm/sec CNT100;
   1:  PR[GP1:91,1] = PR[GP1:90,1] + -6.711;
   1:  PR[GP1:91,2] = PR[GP1:90,2] + 25.688;
   1:L PR[91] R[100]mm/sec CNT100;
   1:  PR[GP1:91,1] = PR[GP1:90,1] + -8.236;
   1:  PR[GP1:91,2] = PR[GP1:90,2] + 25.434;
   1:L PR[91] R[100]mm/sec CNT100;
   1:  PR[GP1:91,1] = PR[GP1:90,1] + -12.952;
   1:  PR[GP1:91,2] = PR[GP1:90,2] + 23.606;
   1:L PR[91] R[100]mm/sec CNT100;
   1:  PR[GP1:91,1] = PR[GP1:90,1] + -14.419;
   1:  PR[GP1:91,2] = PR[GP1:90,2] + 22.955;
   1:L PR[91] R[100]mm/sec CNT100;
   1:  PR[GP1:91,1] = PR[GP1:90,1] + -18.494;
   1:  PR[GP1:91,2] = PR[GP1:90,2] + 20.070;
   1:L PR[91] R[100]mm/sec CNT100;
   1:  PR[GP1:91,1] = PR[GP1:90,1] + -19.804;
   1:  PR[GP1:91,2] = PR[GP1:90,2] + 19.032;
   1:L PR[91] R[100]mm/sec CNT100;
   1:  PR[GP1:91,1] = PR[GP1:90,1] + -22.522;
   1:  PR[GP1:91,2] = PR[GP1:90,2] + 15.986;
   1:L PR[91] R[100]mm/sec CNT100;
   1:  PR[GP1:91,1] = PR[GP1:90,1] + -23.552;
   1:  PR[GP1:91,2] = PR[GP1:90,2] + 14.617;
   1:L PR[91] R[100]mm/sec CNT100;
   1:  PR[GP1:91,1] = PR[GP1:90,1] + -25.514;
   1:  PR[GP1:91,2] = PR[GP1:90,2] + 11.254;
   1:L PR[91] R[100]mm/sec CNT100;
   1:  PR[GP1:91,1] = PR[GP1:90,1] + -26.167;
   1:  PR[GP1:91,2] = PR[GP1:90,2] + 9.664;
   1:L PR[91] R[100]mm/sec CNT100;
   1:  PR[GP1:91,1] = PR[GP1:90,1] + -27.488;
   1:  PR[GP1:91,2] = PR[GP1:90,2] + 5.747;
   1:L PR[91] R[100]mm/sec CNT100;
   1:  PR[GP1:91,1] = PR[GP1:90,1] + -27.710;
   1:  PR[GP1:91,2] = PR[GP1:90,2] + 4.040;
   1:L PR[91] R[100]mm/sec CNT100;
   1:  PR[GP1:91,1] = PR[GP1:90,1] + -28.191;
   1:  PR[GP1:91,2] = PR[GP1:90,2] + -0.298;
   1:L PR[91] R[100]mm/sec CNT100;
   1:  PR[GP1:91,1] = PR[GP1:90,1] + -27.971;
   1:  PR[GP1:91,2] = PR[GP1:90,2] + -1.982;
   1:L PR[91] R[100]mm/sec CNT100;
   1:  PR[GP1:91,1] = PR[GP1:90,1] + -27.538;
   1:  PR[GP1:91,2] = PR[GP1:90,2] + -6.138;
   1:L PR[91] R[100]mm/sec CNT100;
   1:  PR[GP1:91,1] = PR[GP1:90,1] + -26.343;
   1:  PR[GP1:91,2] = PR[GP1:90,2] + -9.894;
   1:L PR[91] R[100]mm/sec CNT100;
   1:  PR[GP1:91,1] = PR[GP1:90,1] + -25.690;
   1:  PR[GP1:91,2] = PR[GP1:90,2] + -11.482;
   1:L PR[91] R[100]mm/sec CNT100;
   1:  PR[GP1:91,1] = PR[GP1:90,1] + -23.725;
   1:  PR[GP1:91,2] = PR[GP1:90,2] + -14.998;
   1:L PR[91] R[100]mm/sec CNT100;
   1:  PR[GP1:91,1] = PR[GP1:90,1] + -22.701;
   1:  PR[GP1:91,2] = PR[GP1:90,2] + -16.357;
   1:L PR[91] R[100]mm/sec CNT100;
   1:  PR[GP1:91,1] = PR[GP1:90,1] + -19.794;
   1:  PR[GP1:91,2] = PR[GP1:90,2] + -19.665;
   1:L PR[91] R[100]mm/sec CNT100;
   1:  PR[GP1:91,1] = PR[GP1:90,1] + -16.410;
   1:  PR[GP1:91,2] = PR[GP1:90,2] + -22.359;
   1:L PR[91] R[100]mm/sec CNT100;
   1:  PR[GP1:91,1] = PR[GP1:90,1] + -14.291;
   1:  PR[GP1:91,2] = PR[GP1:90,2] + -23.648;
   1:L PR[91] R[100]mm/sec CNT100;
   1:  PR[GP1:91,1] = PR[GP1:90,1] + -12.815;
   1:  PR[GP1:91,2] = PR[GP1:90,2] + -24.301;
   1:L PR[91] R[100]mm/sec CNT100;
   1:  PR[GP1:91,1] = PR[GP1:90,1] + -8.081;
   1:  PR[GP1:91,2] = PR[GP1:90,2] + -26.091;
   1:L PR[91] R[100]mm/sec CNT100;
   1:  PR[GP1:91,1] = PR[GP1:90,1] + -6.627;
   1:  PR[GP1:91,2] = PR[GP1:90,2] + -26.332;
   1:L PR[91] R[100]mm/sec CNT100;
   1:  PR[GP1:91,1] = PR[GP1:90,1] + -1.505;
   1:  PR[GP1:91,2] = PR[GP1:90,2] + -26.935;
   1:L PR[91] R[100]mm/sec CNT100;
   1:  PR[GP1:91,1] = PR[GP1:90,1] + -0.062;
   1:  PR[GP1:91,2] = PR[GP1:90,2] + -26.823;
   1:L PR[91] R[100]mm/sec CNT100;
   1:  PR[GP1:91,1] = PR[GP1:90,1] + 0.218;
   1:L PR[91] R[100]mm/sec CNT100;
   1:  PR[GP1:91,1] = PR[GP1:90,1] + 1.704;
   1:  PR[GP1:91,2] = PR[GP1:90,2] + -26.939;
   1:L PR[91] R[100]mm/sec CNT100;
   1:  PR[GP1:91,1] = PR[GP1:90,1] + 4.346;
   1:  PR[GP1:91,2] = PR[GP1:90,2] + -26.781;
   1:L PR[91] R[100]mm/sec CNT100;
   1:  PR[GP1:91,1] = PR[GP1:90,1] + 5.895;
   1:  PR[GP1:91,2] = PR[GP1:90,2] + -26.524;
   1:L PR[91] R[100]mm/sec CNT100;
   1:  PR[GP1:91,1] = PR[GP1:90,1] + 8.426;
   1:  PR[GP1:91,2] = PR[GP1:90,2] + -26.046;
   1:L PR[91] R[100]mm/sec CNT100;
   1:  PR[GP1:91,1] = PR[GP1:90,1] + 13.129;
   1:  PR[GP1:91,2] = PR[GP1:90,2] + -24.217;
   1:L PR[91] R[100]mm/sec CNT100;
   1:  PR[GP1:91,1] = PR[GP1:90,1] + 14.565;
   1:  PR[GP1:91,2] = PR[GP1:90,2] + -23.583;
   1:L PR[91] R[100]mm/sec CNT100;
   1:  PR[GP1:91,1] = PR[GP1:90,1] + 18.647;
   1:  PR[GP1:91,2] = PR[GP1:90,2] + -20.696;
   1:L PR[91] R[100]mm/sec CNT100;
   1:  PR[GP1:91,1] = PR[GP1:90,1] + 19.958;
   1:  PR[GP1:91,2] = PR[GP1:90,2] + -19.659;
   1:L PR[91] R[100]mm/sec CNT100;
   1:  PR[GP1:91,1] = PR[GP1:90,1] + 22.676;
   1:  PR[GP1:91,2] = PR[GP1:90,2] + -16.612;
   1:L PR[91] R[100]mm/sec CNT100;
   1:  PR[GP1:91,1] = PR[GP1:90,1] + 23.708;
   1:  PR[GP1:91,2] = PR[GP1:90,2] + -15.242;
   1:L PR[91] R[100]mm/sec CNT100;
   1:  PR[GP1:91,1] = PR[GP1:90,1] + 25.670;
   1:  PR[GP1:91,2] = PR[GP1:90,2] + -11.878;
   1:L PR[91] R[100]mm/sec CNT100;
   1:  PR[GP1:91,1] = PR[GP1:90,1] + 26.324;
   1:  PR[GP1:91,2] = PR[GP1:90,2] + -10.290;
   1:L PR[91] R[100]mm/sec CNT100;
   1:  PR[GP1:91,1] = PR[GP1:90,1] + 27.644;
   1:  PR[GP1:91,2] = PR[GP1:90,2] + -6.373;
   1:L PR[91] R[100]mm/sec CNT100;
   1:  PR[GP1:91,1] = PR[GP1:90,1] + 27.867;
   1:  PR[GP1:91,2] = PR[GP1:90,2] + -4.664;
   1:L PR[91] R[100]mm/sec CNT100;
   1:  PR[GP1:91,1] = PR[GP1:90,1] + 28.348;
   1:  PR[GP1:91,2] = PR[GP1:90,2] + -0.326;
   1:L PR[91] R[100]mm/sec CNT100;
   1:  PR[GP1:91,1] = PR[GP1:90,1] + 28.128;
   1:  PR[GP1:91,2] = PR[GP1:90,2] + 1.358;
   1:L PR[91] R[100]mm/sec CNT100;
   1:  PR[GP1:91,1] = PR[GP1:90,1] + 27.695;
   1:  PR[GP1:91,2] = PR[GP1:90,2] + 5.513;
   1:L PR[91] R[100]mm/sec CNT100;
   1:  PR[GP1:91,1] = PR[GP1:90,1] + 26.501;
   1:  PR[GP1:91,2] = PR[GP1:90,2] + 9.269;
   1:L PR[91] R[100]mm/sec CNT100;
   1:  PR[GP1:91,1] = PR[GP1:90,1] + 25.849;
   1:  PR[GP1:91,2] = PR[GP1:90,2] + 10.853;
   1:L PR[91] R[100]mm/sec CNT100;
   1:  PR[GP1:91,1] = PR[GP1:90,1] + 23.884;
   1:  PR[GP1:91,2] = PR[GP1:90,2] + 14.370;
   1:L PR[91] R[100]mm/sec CNT100;
   1:  PR[GP1:91,1] = PR[GP1:90,1] + 22.861;
   1:  PR[GP1:91,2] = PR[GP1:90,2] + 15.729;
   1:L PR[91] R[100]mm/sec CNT100;
   1:  PR[GP1:91,1] = PR[GP1:90,1] + 19.957;
   1:  PR[GP1:91,2] = PR[GP1:90,2] + 19.035;
   1:L PR[91] R[100]mm/sec CNT100;
   1:  PR[GP1:91,1] = PR[GP1:90,1] + 18.652;
   1:  PR[GP1:91,2] = PR[GP1:90,2] + 20.069;
   1:L PR[91] R[100]mm/sec CNT100;
   1:  PR[GP1:91,1] = PR[GP1:90,1] + 14.576;
   1:  PR[GP1:91,2] = PR[GP1:90,2] + 22.955;
   1:L PR[91] R[100]mm/sec CNT100;
   1:  PR[GP1:91,1] = PR[GP1:90,1] + 13.109;
   1:  PR[GP1:91,2] = PR[GP1:90,2] + 23.606;
   1:L PR[91] R[100]mm/sec CNT100;
   1:  PR[GP1:91,1] = PR[GP1:90,1] + 8.392;
   1:  PR[GP1:91,2] = PR[GP1:90,2] + 25.434;
   1:L PR[91] R[100]mm/sec CNT100;
   1:  PR[GP1:91,1] = PR[GP1:90,1] + 6.867;
   1:  PR[GP1:91,2] = PR[GP1:90,2] + 25.688;
   1:L PR[91] R[100]mm/sec CNT100;
   1:  PR[GP1:91,1] = PR[GP1:90,1] + 1.772;
   1:  PR[GP1:91,2] = PR[GP1:90,2] + 26.319;
   1:L PR[91] R[100]mm/sec CNT100;
   1:  PR[GP1:91,1] = PR[GP1:90,1] + 0.214;
   1:  PR[GP1:91,2] = PR[GP1:90,2] + 26.203;
   1:L PR[91] R[100]mm/sec CNT100;
   1:  PR[91] = PR[90];
   1:  PR[GP1:91,1] = PR[GP1:90,1] + -1.354;
   1:  PR[GP1:91,2] = PR[GP1:90,2] + 26.457;
   1:  PR[GP1:91,3] = PR[GP1:90,3] + 71.065;
   1:L PR[91] R[100]mm/sec CNT100;
   1:  PR[GP1:91,1] = PR[GP1:90,1] + -6.723;
   1:  PR[GP1:91,2] = PR[GP1:90,2] + 25.792;
   1:L PR[91] R[100]mm/sec CNT100;
   1:  PR[GP1:91,1] = PR[GP1:90,1] + -7.994;
   1:  PR[GP1:91,2] = PR[GP1:90,2] + 25.580;
   1:L PR[91] R[100]mm/sec CNT100;
   1:  PR[GP1:91,1] = PR[GP1:90,1] + -12.973;
   1:  PR[GP1:91,2] = PR[GP1:90,2] + 23.651;
   1:L PR[91] R[100]mm/sec CNT100;
   1:  PR[GP1:91,1] = PR[GP1:90,1] + -14.197;
   1:  PR[GP1:91,2] = PR[GP1:90,2] + 23.108;
   1:L PR[91] R[100]mm/sec CNT100;
   1:  PR[GP1:91,1] = PR[GP1:90,1] + -18.510;
   1:  PR[GP1:91,2] = PR[GP1:90,2] + 20.054;
   1:L PR[91] R[100]mm/sec CNT100;
   1:  PR[GP1:91,1] = PR[GP1:90,1] + -19.605;
   1:  PR[GP1:91,2] = PR[GP1:90,2] + 19.186;
   1:L PR[91] R[100]mm/sec CNT100;
   1:  PR[GP1:91,1] = PR[GP1:90,1] + -22.490;
   1:  PR[GP1:91,2] = PR[GP1:90,2] + 15.953;
   1:L PR[91] R[100]mm/sec CNT100;
   1:  PR[GP1:91,1] = PR[GP1:90,1] + -23.350;
   1:  PR[GP1:91,2] = PR[GP1:90,2] + 14.810;
   1:L PR[91] R[100]mm/sec CNT100;
   1:  PR[GP1:91,1] = PR[GP1:90,1] + -25.436;
   1:  PR[GP1:91,2] = PR[GP1:90,2] + 11.234;
   1:L PR[91] R[100]mm/sec CNT100;
   1:  PR[GP1:91,1] = PR[GP1:90,1] + -25.979;
   1:  PR[GP1:91,2] = PR[GP1:90,2] + 9.911;
   1:L PR[91] R[100]mm/sec CNT100;
   1:  PR[GP1:91,1] = PR[GP1:90,1] + -27.386;
   1:  PR[GP1:91,2] = PR[GP1:90,2] + 5.740;
   1:L PR[91] R[100]mm/sec CNT100;
   1:  PR[GP1:91,1] = PR[GP1:90,1] + -27.570;
   1:  PR[GP1:91,2] = PR[GP1:90,2] + 4.324;
   1:L PR[91] R[100]mm/sec CNT100;
   1:  PR[GP1:91,1] = PR[GP1:90,1] + -28.082;
   1:  PR[GP1:91,2] = PR[GP1:90,2] + -0.298;
   1:L PR[91] R[100]mm/sec CNT100;
   1:  PR[GP1:91,1] = PR[GP1:90,1] + -27.900;
   1:  PR[GP1:91,2] = PR[GP1:90,2] + -1.693;
   1:L PR[91] R[100]mm/sec CNT100;
   1:  PR[GP1:91,1] = PR[GP1:90,1] + -27.439;
   1:  PR[GP1:91,2] = PR[GP1:90,2] + -6.115;
   1:L PR[91] R[100]mm/sec CNT100;
   1:  PR[GP1:91,1] = PR[GP1:90,1] + -26.167;
   1:  PR[GP1:91,2] = PR[GP1:90,2] + -10.116;
   1:L PR[91] R[100]mm/sec CNT100;
   1:  PR[GP1:91,1] = PR[GP1:90,1] + -25.624;
   1:  PR[GP1:91,2] = PR[GP1:90,2] + -11.436;
   1:L PR[91] R[100]mm/sec CNT100;
   1:  PR[GP1:91,1] = PR[GP1:90,1] + -23.534;
   1:  PR[GP1:91,2] = PR[GP1:90,2] + -15.175;
   1:L PR[91] R[100]mm/sec CNT100;
   1:  PR[GP1:91,1] = PR[GP1:90,1] + -22.680;
   1:  PR[GP1:91,2] = PR[GP1:90,2] + -16.309;
   1:L PR[91] R[100]mm/sec CNT100;
   1:  PR[GP1:91,1] = PR[GP1:90,1] + -19.596;
   1:  PR[GP1:91,2] = PR[GP1:90,2] + -19.818;
   1:L PR[91] R[100]mm/sec CNT100;
   1:  PR[GP1:91,1] = PR[GP1:90,1] + -16.307;
   1:  PR[GP1:91,2] = PR[GP1:90,2] + -22.438;
   1:L PR[91] R[100]mm/sec CNT100;
   1:  PR[GP1:91,1] = PR[GP1:90,1] + -14.061;
   1:  PR[GP1:91,2] = PR[GP1:90,2] + -23.805;
   1:L PR[91] R[100]mm/sec CNT100;
   1:  PR[GP1:91,1] = PR[GP1:90,1] + -12.830;
   1:  PR[GP1:91,2] = PR[GP1:90,2] + -24.349;
   1:L PR[91] R[100]mm/sec CNT100;
   1:  PR[GP1:91,1] = PR[GP1:90,1] + -7.832;
   1:  PR[GP1:91,2] = PR[GP1:90,2] + -26.239;
   1:L PR[91] R[100]mm/sec CNT100;
   1:  PR[GP1:91,1] = PR[GP1:90,1] + -6.636;
   1:  PR[GP1:91,2] = PR[GP1:90,2] + -26.437;
   1:L PR[91] R[100]mm/sec CNT100;
   1:  PR[GP1:91,1] = PR[GP1:90,1] + -1.243;
   1:  PR[GP1:91,2] = PR[GP1:90,2] + -27.073;
   1:L PR[91] R[100]mm/sec CNT100;
   1:  PR[GP1:91,1] = PR[GP1:90,1] + 0.001;
   1:  PR[GP1:91,2] = PR[GP1:90,2] + -26.976;
   1:L PR[91] R[100]mm/sec CNT100;
   1:  PR[GP1:91,1] = PR[GP1:90,1] + 1.436;
   1:  PR[GP1:91,2] = PR[GP1:90,2] + -27.076;
   1:L PR[91] R[100]mm/sec CNT100;
   1:  PR[GP1:91,1] = PR[GP1:90,1] + 4.229;
   1:  PR[GP1:91,2] = PR[GP1:90,2] + -26.909;
   1:L PR[91] R[100]mm/sec CNT100;
   1:  PR[GP1:91,1] = PR[GP1:90,1] + 5.514;
   1:  PR[GP1:91,2] = PR[GP1:90,2] + -26.696;
   1:L PR[91] R[100]mm/sec CNT100;
   1:  PR[GP1:91,1] = PR[GP1:90,1] + 8.188;
   1:  PR[GP1:91,2] = PR[GP1:90,2] + -26.191;
   1:L PR[91] R[100]mm/sec CNT100;
   1:  PR[GP1:91,1] = PR[GP1:90,1] + 13.152;
   1:  PR[GP1:91,2] = PR[GP1:90,2] + -24.261;
   1:L PR[91] R[100]mm/sec CNT100;
   1:  PR[GP1:91,1] = PR[GP1:90,1] + 14.343;
   1:  PR[GP1:91,2] = PR[GP1:90,2] + -23.735;
   1:L PR[91] R[100]mm/sec CNT100;
   1:  PR[GP1:91,1] = PR[GP1:90,1] + 18.663;
   1:  PR[GP1:91,2] = PR[GP1:90,2] + -20.680;
   1:L PR[91] R[100]mm/sec CNT100;
   1:  PR[GP1:91,1] = PR[GP1:90,1] + 19.760;
   1:  PR[GP1:91,2] = PR[GP1:90,2] + -19.812;
   1:L PR[91] R[100]mm/sec CNT100;
   1:  PR[GP1:91,1] = PR[GP1:90,1] + 22.644;
   1:  PR[GP1:91,2] = PR[GP1:90,2] + -16.579;
   1:L PR[91] R[100]mm/sec CNT100;
   1:  PR[GP1:91,1] = PR[GP1:90,1] + 23.506;
   1:  PR[GP1:91,2] = PR[GP1:90,2] + -15.435;
   1:L PR[91] R[100]mm/sec CNT100;
   1:  PR[GP1:91,1] = PR[GP1:90,1] + 25.592;
   1:  PR[GP1:91,2] = PR[GP1:90,2] + -11.858;
   1:L PR[91] R[100]mm/sec CNT100;
   1:  PR[GP1:91,1] = PR[GP1:90,1] + 26.136;
   1:  PR[GP1:91,2] = PR[GP1:90,2] + -10.536;
   1:L PR[91] R[100]mm/sec CNT100;
   1:  PR[GP1:91,1] = PR[GP1:90,1] + 27.542;
   1:  PR[GP1:91,2] = PR[GP1:90,2] + -6.366;
   1:L PR[91] R[100]mm/sec CNT100;
   1:  PR[GP1:91,1] = PR[GP1:90,1] + 27.727;
   1:  PR[GP1:91,2] = PR[GP1:90,2] + -4.948;
   1:L PR[91] R[100]mm/sec CNT100;
   1:  PR[GP1:91,1] = PR[GP1:90,1] + 28.239;
   1:  PR[GP1:91,2] = PR[GP1:90,2] + -0.326;
   1:L PR[91] R[100]mm/sec CNT100;
   1:  PR[GP1:91,1] = PR[GP1:90,1] + 28.058;
   1:  PR[GP1:91,2] = PR[GP1:90,2] + 1.069;
   1:L PR[91] R[100]mm/sec CNT100;
   1:  PR[GP1:91,1] = PR[GP1:90,1] + 27.597;
   1:  PR[GP1:91,2] = PR[GP1:90,2] + 5.490;
   1:L PR[91] R[100]mm/sec CNT100;
   1:  PR[GP1:91,1] = PR[GP1:90,1] + 26.325;
   1:  PR[GP1:91,2] = PR[GP1:90,2] + 9.490;
   1:L PR[91] R[100]mm/sec CNT100;
   1:  PR[GP1:91,1] = PR[GP1:90,1] + 25.783;
   1:  PR[GP1:91,2] = PR[GP1:90,2] + 10.808;
   1:L PR[91] R[100]mm/sec CNT100;
   1:  PR[GP1:91,1] = PR[GP1:90,1] + 23.693;
   1:  PR[GP1:91,2] = PR[GP1:90,2] + 14.548;
   1:L PR[91] R[100]mm/sec CNT100;
   1:  PR[GP1:91,1] = PR[GP1:90,1] + 22.840;
   1:  PR[GP1:91,2] = PR[GP1:90,2] + 15.681;
   1:L PR[91] R[100]mm/sec CNT100;
   1:  PR[GP1:91,1] = PR[GP1:90,1] + 19.758;
   1:  PR[GP1:91,2] = PR[GP1:90,2] + 19.189;
   1:L PR[91] R[100]mm/sec CNT100;
   1:  PR[GP1:91,1] = PR[GP1:90,1] + 18.667;
   1:  PR[GP1:91,2] = PR[GP1:90,2] + 20.053;
   1:L PR[91] R[100]mm/sec CNT100;
   1:  PR[GP1:91,1] = PR[GP1:90,1] + 14.354;
   1:  PR[GP1:91,2] = PR[GP1:90,2] + 23.108;
   1:L PR[91] R[100]mm/sec CNT100;
   1:  PR[GP1:91,1] = PR[GP1:90,1] + 13.130;
   1:  PR[GP1:91,2] = PR[GP1:90,2] + 23.650;
   1:L PR[91] R[100]mm/sec CNT100;
   1:  PR[GP1:91,1] = PR[GP1:90,1] + 8.150;
   1:  PR[GP1:91,2] = PR[GP1:90,2] + 25.580;
   1:L PR[91] R[100]mm/sec CNT100;
   1:  PR[GP1:91,1] = PR[GP1:90,1] + 6.879;
   1:  PR[GP1:91,2] = PR[GP1:90,2] + 25.792;
   1:L PR[91] R[100]mm/sec CNT100;
   1:  PR[GP1:91,1] = PR[GP1:90,1] + 1.514;
   1:  PR[GP1:91,2] = PR[GP1:90,2] + 26.457;
   1:L PR[91] R[100]mm/sec CNT100;
   1:  PR[GP1:91,1] = PR[GP1:90,1] + 0.153;
   1:  PR[GP1:91,2] = PR[GP1:90,2] + 26.355;
   1:L PR[91] R[100]mm/sec CNT100;
   1:  PR[91] = PR[90];
   1:  PR[GP1:91,1] = PR[GP1:90,1] + -1.096;
   1:  PR[GP1:91,2] = PR[GP1:90,2] + 26.595;
   1:  PR[GP1:91,3] = PR[GP1:90,3] + 71.675;
   1:L PR[91] R[100]mm/sec CNT100;
   1:  PR[GP1:91,1] = PR[GP1:90,1] + -6.735;
   1:  PR[GP1:91,2] = PR[GP1:90,2] + 25.896;
   1:L PR[91] R[100]mm/sec CNT100;
   1:  PR[GP1:91,1] = PR[GP1:90,1] + -7.753;
   1:  PR[GP1:91,2] = PR[GP1:90,2] + 25.726;
   1:L PR[91] R[100]mm/sec CNT100;
   1:  PR[GP1:91,1] = PR[GP1:90,1] + -12.994;
   1:  PR[GP1:91,2] = PR[GP1:90,2] + 23.695;
   1:L PR[91] R[100]mm/sec CNT100;
   1:  PR[GP1:91,1] = PR[GP1:90,1] + -13.975;
   1:  PR[GP1:91,2] = PR[GP1:90,2] + 23.260;
   1:L PR[91] R[100]mm/sec CNT100;
   1:  PR[GP1:91,1] = PR[GP1:90,1] + -18.525;
   1:  PR[GP1:91,2] = PR[GP1:90,2] + 20.038;
   1:L PR[91] R[100]mm/sec CNT100;
   1:  PR[GP1:91,1] = PR[GP1:90,1] + -19.406;
   1:  PR[GP1:91,2] = PR[GP1:90,2] + 19.340;
   1:L PR[91] R[100]mm/sec CNT100;
   1:  PR[GP1:91,1] = PR[GP1:90,1] + -22.457;
   1:  PR[GP1:91,2] = PR[GP1:90,2] + 15.921;
   1:L PR[91] R[100]mm/sec CNT100;
   1:  PR[GP1:91,1] = PR[GP1:90,1] + -23.148;
   1:  PR[GP1:91,2] = PR[GP1:90,2] + 15.004;
   1:L PR[91] R[100]mm/sec CNT100;
   1:  PR[GP1:91,1] = PR[GP1:90,1] + -25.358;
   1:  PR[GP1:91,2] = PR[GP1:90,2] + 11.214;
   1:L PR[91] R[100]mm/sec CNT100;
   1:  PR[GP1:91,1] = PR[GP1:90,1] + -25.792;
   1:  PR[GP1:91,2] = PR[GP1:90,2] + 10.158;
   1:L PR[91] R[100]mm/sec CNT100;
   1:  PR[GP1:91,1] = PR[GP1:90,1] + -27.284;
   1:  PR[GP1:91,2] = PR[GP1:90,2] + 5.733;
   1:L PR[91] R[100]mm/sec CNT100;
   1:  PR[GP1:91,1] = PR[GP1:90,1] + -27.430;
   1:  PR[GP1:91,2] = PR[GP1:90,2] + 4.609;
   1:L PR[91] R[100]mm/sec CNT100;
   1:  PR[GP1:91,1] = PR[GP1:90,1] + -27.974;
   1:  PR[GP1:91,2] = PR[GP1:90,2] + -0.298;
   1:L PR[91] R[100]mm/sec CNT100;
   1:  PR[GP1:91,1] = PR[GP1:90,1] + -27.830;
   1:  PR[GP1:91,2] = PR[GP1:90,2] + -1.405;
   1:L PR[91] R[100]mm/sec CNT100;
   1:  PR[GP1:91,1] = PR[GP1:90,1] + -27.341;
   1:  PR[GP1:91,2] = PR[GP1:90,2] + -6.092;
   1:L PR[91] R[100]mm/sec CNT100;
   1:  PR[GP1:91,1] = PR[GP1:90,1] + -25.991;
   1:  PR[GP1:91,2] = PR[GP1:90,2] + -10.337;
   1:L PR[91] R[100]mm/sec CNT100;
   1:  PR[GP1:91,1] = PR[GP1:90,1] + -25.557;
   1:  PR[GP1:91,2] = PR[GP1:90,2] + -11.391;
   1:L PR[91] R[100]mm/sec CNT100;
   1:  PR[GP1:91,1] = PR[GP1:90,1] + -23.343;
   1:  PR[GP1:91,2] = PR[GP1:90,2] + -15.353;
   1:L PR[91] R[100]mm/sec CNT100;
   1:  PR[GP1:91,1] = PR[GP1:90,1] + -22.659;
   1:  PR[GP1:91,2] = PR[GP1:90,2] + -16.260;
   1:L PR[91] R[100]mm/sec CNT100;
   1:  PR[GP1:91,1] = PR[GP1:90,1] + -19.398;
   1:  PR[GP1:91,2] = PR[GP1:90,2] + -19.972;
   1:L PR[91] R[100]mm/sec CNT100;
   1:  PR[GP1:91,1] = PR[GP1:90,1] + -16.204;
   1:  PR[GP1:91,2] = PR[GP1:90,2] + -22.517;
   1:L PR[91] R[100]mm/sec CNT100;
   1:  PR[GP1:91,1] = PR[GP1:90,1] + -13.830;
   1:  PR[GP1:91,2] = PR[GP1:90,2] + -23.962;
   1:L PR[91] R[100]mm/sec CNT100;
   1:  PR[GP1:91,1] = PR[GP1:90,1] + -12.845;
   1:  PR[GP1:91,2] = PR[GP1:90,2] + -24.398;
   1:L PR[91] R[100]mm/sec CNT100;
   1:  PR[GP1:91,1] = PR[GP1:90,1] + -7.584;
   1:  PR[GP1:91,2] = PR[GP1:90,2] + -26.387;
   1:L PR[91] R[100]mm/sec CNT100;
   1:  PR[GP1:91,1] = PR[GP1:90,1] + -6.645;
   1:  PR[GP1:91,2] = PR[GP1:90,2] + -26.542;
   1:L PR[91] R[100]mm/sec CNT100;
   1:  PR[GP1:91,1] = PR[GP1:90,1] + -0.981;
   1:  PR[GP1:91,2] = PR[GP1:90,2] + -27.210;
   1:L PR[91] R[100]mm/sec CNT100;
   1:  PR[GP1:91,1] = PR[GP1:90,1] + 0.014;
   1:  PR[GP1:91,2] = PR[GP1:90,2] + -27.132;
   1:L PR[91] R[100]mm/sec CNT100;
   1:  PR[GP1:91,1] = PR[GP1:90,1] + 1.174;
   1:  PR[GP1:91,2] = PR[GP1:90,2] + -27.213;
   1:L PR[91] R[100]mm/sec CNT100;
   1:  PR[GP1:91,1] = PR[GP1:90,1] + 4.111;
   1:  PR[GP1:91,2] = PR[GP1:90,2] + -27.038;
   1:L PR[91] R[100]mm/sec CNT100;
   1:  PR[GP1:91,1] = PR[GP1:90,1] + 5.133;
   1:  PR[GP1:91,2] = PR[GP1:90,2] + -26.868;
   1:L PR[91] R[100]mm/sec CNT100;
   1:  PR[GP1:91,1] = PR[GP1:90,1] + 7.951;
   1:  PR[GP1:91,2] = PR[GP1:90,2] + -26.336;
   1:L PR[91] R[100]mm/sec CNT100;
   1:  PR[GP1:91,1] = PR[GP1:90,1] + 13.176;
   1:  PR[GP1:91,2] = PR[GP1:90,2] + -24.305;
   1:L PR[91] R[100]mm/sec CNT100;
   1:  PR[GP1:91,1] = PR[GP1:90,1] + 14.121;
   1:  PR[GP1:91,2] = PR[GP1:90,2] + -23.886;
   1:L PR[91] R[100]mm/sec CNT100;
   1:  PR[GP1:91,1] = PR[GP1:90,1] + 18.679;
   1:  PR[GP1:91,2] = PR[GP1:90,2] + -20.663;
   1:L PR[91] R[100]mm/sec CNT100;
   1:  PR[GP1:91,1] = PR[GP1:90,1] + 19.561;
   1:  PR[GP1:91,2] = PR[GP1:90,2] + -19.966;
   1:L PR[91] R[100]mm/sec CNT100;
   1:  PR[GP1:91,1] = PR[GP1:90,1] + 22.613;
   1:  PR[GP1:91,2] = PR[GP1:90,2] + -16.546;
   1:L PR[91] R[100]mm/sec CNT100;
   1:  PR[GP1:91,1] = PR[GP1:90,1] + 23.304;
   1:  PR[GP1:91,2] = PR[GP1:90,2] + -15.628;
   1:L PR[91] R[100]mm/sec CNT100;
   1:  PR[GP1:91,1] = PR[GP1:90,1] + 25.515;
   1:  PR[GP1:91,2] = PR[GP1:90,2] + -11.837;
   1:L PR[91] R[100]mm/sec CNT100;
   1:  PR[GP1:91,1] = PR[GP1:90,1] + 25.949;
   1:  PR[GP1:91,2] = PR[GP1:90,2] + -10.782;
   1:L PR[91] R[100]mm/sec CNT100;
   1:  PR[GP1:91,1] = PR[GP1:90,1] + 27.440;
   1:  PR[GP1:91,2] = PR[GP1:90,2] + -6.359;
   1:L PR[91] R[100]mm/sec CNT100;
   1:  PR[GP1:91,1] = PR[GP1:90,1] + 27.587;
   1:  PR[GP1:91,2] = PR[GP1:90,2] + -5.232;
   1:L PR[91] R[100]mm/sec CNT100;
   1:  PR[GP1:91,1] = PR[GP1:90,1] + 28.131;
   1:  PR[GP1:91,2] = PR[GP1:90,2] + -0.326;
   1:L PR[91] R[100]mm/sec CNT100;
   1:  PR[GP1:91,1] = PR[GP1:90,1] + 27.987;
   1:  PR[GP1:91,2] = PR[GP1:90,2] + 0.781;
   1:L PR[91] R[100]mm/sec CNT100;
   1:  PR[GP1:91,1] = PR[GP1:90,1] + 27.498;
   1:  PR[GP1:91,2] = PR[GP1:90,2] + 5.467;
   1:L PR[91] R[100]mm/sec CNT100;
   1:  PR[GP1:91,1] = PR[GP1:90,1] + 26.148;
   1:  PR[GP1:91,2] = PR[GP1:90,2] + 9.712;
   1:L PR[91] R[100]mm/sec CNT100;
   1:  PR[GP1:91,1] = PR[GP1:90,1] + 25.716;
   1:  PR[GP1:91,2] = PR[GP1:90,2] + 10.763;
   1:L PR[91] R[100]mm/sec CNT100;
   1:  PR[GP1:91,1] = PR[GP1:90,1] + 23.502;
   1:  PR[GP1:91,2] = PR[GP1:90,2] + 14.725;
   1:L PR[91] R[100]mm/sec CNT100;
   1:  PR[GP1:91,1] = PR[GP1:90,1] + 22.819;
   1:  PR[GP1:91,2] = PR[GP1:90,2] + 15.633;
   1:L PR[91] R[100]mm/sec CNT100;
   1:  PR[GP1:91,1] = PR[GP1:90,1] + 19.559;
   1:  PR[GP1:91,2] = PR[GP1:90,2] + 19.343;
   1:L PR[91] R[100]mm/sec CNT100;
   1:  PR[GP1:91,1] = PR[GP1:90,1] + 18.683;
   1:  PR[GP1:91,2] = PR[GP1:90,2] + 20.037;
   1:L PR[91] R[100]mm/sec CNT100;
   1:  PR[GP1:91,1] = PR[GP1:90,1] + 14.132;
   1:  PR[GP1:91,2] = PR[GP1:90,2] + 23.260;
   1:L PR[91] R[100]mm/sec CNT100;
   1:  PR[GP1:91,1] = PR[GP1:90,1] + 13.151;
   1:  PR[GP1:91,2] = PR[GP1:90,2] + 23.695;
   1:L PR[91] R[100]mm/sec CNT100;
   1:  PR[GP1:91,1] = PR[GP1:90,1] + 7.909;
   1:  PR[GP1:91,2] = PR[GP1:90,2] + 25.726;
   1:L PR[91] R[100]mm/sec CNT100;
   1:  PR[GP1:91,1] = PR[GP1:90,1] + 6.891;
   1:  PR[GP1:91,2] = PR[GP1:90,2] + 25.896;
   1:L PR[91] R[100]mm/sec CNT100;
   1:  PR[GP1:91,1] = PR[GP1:90,1] + 1.256;
   1:  PR[GP1:91,2] = PR[GP1:90,2] + 26.594;
   1:L PR[91] R[100]mm/sec CNT100;
   1:  PR[GP1:91,1] = PR[GP1:90,1] + 0.141;
   1:  PR[GP1:91,2] = PR[GP1:90,2] + 26.511;
   1:L PR[91] R[100]mm/sec CNT100;
   1:  PR[91] = PR[90];
   1:  PR[GP1:91,1] = PR[GP1:90,1] + -0.838;
   1:  PR[GP1:91,2] = PR[GP1:90,2] + 26.732;
   1:  PR[GP1:91,3] = PR[GP1:90,3] + 72.285;
   1:L PR[91] R[100]mm/sec CNT100;
   1:  PR[GP1:91,1] = PR[GP1:90,1] + -6.747;
   1:  PR[GP1:91,2] = PR[GP1:90,2] + 26.000;
   1:L PR[91] R[100]mm/sec CNT100;
   1:  PR[GP1:91,1] = PR[GP1:90,1] + -7.511;
   1:  PR[GP1:91,2] = PR[GP1:90,2] + 25.873;
   1:L PR[91] R[100]mm/sec CNT100;
   1:  PR[GP1:91,1] = PR[GP1:90,1] + -13.015;
   1:  PR[GP1:91,2] = PR[GP1:90,2] + 23.740;
   1:L PR[91] R[100]mm/sec CNT100;
   1:  PR[GP1:91,1] = PR[GP1:90,1] + -13.753;
   1:  PR[GP1:91,2] = PR[GP1:90,2] + 23.413;
   1:L PR[91] R[100]mm/sec CNT100;
   1:  PR[GP1:91,1] = PR[GP1:90,1] + -18.541;
   1:  PR[GP1:91,2] = PR[GP1:90,2] + 20.022;
   1:L PR[91] R[100]mm/sec CNT100;
   1:  PR[GP1:91,1] = PR[GP1:90,1] + -19.207;
   1:  PR[GP1:91,2] = PR[GP1:90,2] + 19.494;
   1:L PR[91] R[100]mm/sec CNT100;
   1:  PR[GP1:91,1] = PR[GP1:90,1] + -22.425;
   1:  PR[GP1:91,2] = PR[GP1:90,2] + 15.888;
   1:L PR[91] R[100]mm/sec CNT100;
   1:  PR[GP1:91,1] = PR[GP1:90,1] + -22.945;
   1:  PR[GP1:91,2] = PR[GP1:90,2] + 15.197;
   1:L PR[91] R[100]mm/sec CNT100;
   1:  PR[GP1:91,1] = PR[GP1:90,1] + -25.280;
   1:  PR[GP1:91,2] = PR[GP1:90,2] + 11.194;
   1:L PR[91] R[100]mm/sec CNT100;
   1:  PR[GP1:91,1] = PR[GP1:90,1] + -25.604;
   1:  PR[GP1:91,2] = PR[GP1:90,2] + 10.405;
   1:L PR[91] R[100]mm/sec CNT100;
   1:  PR[GP1:91,1] = PR[GP1:90,1] + -27.182;
   1:  PR[GP1:91,2] = PR[GP1:90,2] + 5.727;
   1:L PR[91] R[100]mm/sec CNT100;
   1:  PR[GP1:91,1] = PR[GP1:90,1] + -27.290;
   1:  PR[GP1:91,2] = PR[GP1:90,2] + 4.893;
   1:L PR[91] R[100]mm/sec CNT100;
   1:  PR[GP1:91,1] = PR[GP1:90,1] + -27.866;
   1:  PR[GP1:91,2] = PR[GP1:90,2] + -0.298;
   1:L PR[91] R[100]mm/sec CNT100;
   1:  PR[GP1:91,1] = PR[GP1:90,1] + -27.759;
   1:  PR[GP1:91,2] = PR[GP1:90,2] + -1.116;
   1:L PR[91] R[100]mm/sec CNT100;
   1:  PR[GP1:91,1] = PR[GP1:90,1] + -27.242;
   1:  PR[GP1:91,2] = PR[GP1:90,2] + -6.068;
   1:L PR[91] R[100]mm/sec CNT100;
   1:  PR[GP1:91,1] = PR[GP1:90,1] + -25.814;
   1:  PR[GP1:91,2] = PR[GP1:90,2] + -10.558;
   1:L PR[91] R[100]mm/sec CNT100;
   1:  PR[GP1:91,1] = PR[GP1:90,1] + -25.491;
   1:  PR[GP1:91,2] = PR[GP1:90,2] + -11.346;
   1:L PR[91] R[100]mm/sec CNT100;
   1:  PR[GP1:91,1] = PR[GP1:90,1] + -23.152;
   1:  PR[GP1:91,2] = PR[GP1:90,2] + -15.530;
   1:L PR[91] R[100]mm/sec CNT100;
   1:  PR[GP1:91,1] = PR[GP1:90,1] + -22.638;
   1:  PR[GP1:91,2] = PR[GP1:90,2] + -16.212;
   1:L PR[91] R[100]mm/sec CNT100;
   1:  PR[GP1:91,1] = PR[GP1:90,1] + -19.199;
   1:  PR[GP1:91,2] = PR[GP1:90,2] + -20.126;
   1:L PR[91] R[100]mm/sec CNT100;
   1:  PR[GP1:91,1] = PR[GP1:90,1] + -16.101;
   1:  PR[GP1:91,2] = PR[GP1:90,2] + -22.596;
   1:L PR[91] R[100]mm/sec CNT100;
   1:  PR[GP1:91,1] = PR[GP1:90,1] + -13.599;
   1:  PR[GP1:91,2] = PR[GP1:90,2] + -24.119;
   1:L PR[91] R[100]mm/sec CNT100;
   1:  PR[GP1:91,1] = PR[GP1:90,1] + -12.860;
   1:  PR[GP1:91,2] = PR[GP1:90,2] + -24.446;
   1:L PR[91] R[100]mm/sec CNT100;
   1:  PR[GP1:91,1] = PR[GP1:90,1] + -7.335;
   1:  PR[GP1:91,2] = PR[GP1:90,2] + -26.535;
   1:L PR[91] R[100]mm/sec CNT100;
   1:  PR[GP1:91,1] = PR[GP1:90,1] + -6.655;
   1:  PR[GP1:91,2] = PR[GP1:90,2] + -26.647;
   1:L PR[91] R[100]mm/sec CNT100;
   1:  PR[GP1:91,1] = PR[GP1:90,1] + -0.719;
   1:  PR[GP1:91,2] = PR[GP1:90,2] + -27.347;
   1:L PR[91] R[100]mm/sec CNT100;
   1:  PR[GP1:91,1] = PR[GP1:90,1] + 0.026;
   1:  PR[GP1:91,2] = PR[GP1:90,2] + -27.289;
   1:L PR[91] R[100]mm/sec CNT100;
   1:  PR[GP1:91,1] = PR[GP1:90,1] + 0.912;
   1:  PR[GP1:91,2] = PR[GP1:90,2] + -27.350;
   1:L PR[91] R[100]mm/sec CNT100;
   1:  PR[GP1:91,1] = PR[GP1:90,1] + 3.993;
   1:  PR[GP1:91,2] = PR[GP1:90,2] + -27.166;
   1:L PR[91] R[100]mm/sec CNT100;
   1:  PR[GP1:91,1] = PR[GP1:90,1] + 4.751;
   1:  PR[GP1:91,2] = PR[GP1:90,2] + -27.040;
   1:L PR[91] R[100]mm/sec CNT100;
   1:  PR[GP1:91,1] = PR[GP1:90,1] + 7.713;
   1:  PR[GP1:91,2] = PR[GP1:90,2] + -26.481;
   1:L PR[91] R[100]mm/sec CNT100;
   1:  PR[GP1:91,1] = PR[GP1:90,1] + 13.199;
   1:  PR[GP1:91,2] = PR[GP1:90,2] + -24.348;
   1:L PR[91] R[100]mm/sec CNT100;
   1:  PR[GP1:91,1] = PR[GP1:90,1] + 13.899;
   1:  PR[GP1:91,2] = PR[GP1:90,2] + -24.038;
   1:L PR[91] R[100]mm/sec CNT100;
   1:  PR[GP1:91,1] = PR[GP1:90,1] + 18.696;
   1:  PR[GP1:91,2] = PR[GP1:90,2] + -20.647;
   1:L PR[91] R[100]mm/sec CNT100;
   1:  PR[GP1:91,1] = PR[GP1:90,1] + 19.363;
   1:  PR[GP1:91,2] = PR[GP1:90,2] + -20.119;
   1:L PR[91] R[100]mm/sec CNT100;
   1:  PR[GP1:91,1] = PR[GP1:90,1] + 22.581;
   1:  PR[GP1:91,2] = PR[GP1:90,2] + -16.512;
   1:L PR[91] R[100]mm/sec CNT100;
   1:  PR[GP1:91,1] = PR[GP1:90,1] + 23.102;
   1:  PR[GP1:91,2] = PR[GP1:90,2] + -15.821;
   1:L PR[91] R[100]mm/sec CNT100;
   1:  PR[GP1:91,1] = PR[GP1:90,1] + 25.437;
   1:  PR[GP1:91,2] = PR[GP1:90,2] + -11.817;
   1:L PR[91] R[100]mm/sec CNT100;
   1:  PR[GP1:91,1] = PR[GP1:90,1] + 25.762;
   1:  PR[GP1:91,2] = PR[GP1:90,2] + -11.028;
   1:L PR[91] R[100]mm/sec CNT100;
   1:  PR[GP1:91,1] = PR[GP1:90,1] + 27.338;
   1:  PR[GP1:91,2] = PR[GP1:90,2] + -6.352;
   1:L PR[91] R[100]mm/sec CNT100;
   1:  PR[GP1:91,1] = PR[GP1:90,1] + 27.447;
   1:  PR[GP1:91,2] = PR[GP1:90,2] + -5.516;
   1:L PR[91] R[100]mm/sec CNT100;
   1:  PR[GP1:91,1] = PR[GP1:90,1] + 28.022;
   1:  PR[GP1:91,2] = PR[GP1:90,2] + -0.326;
   1:L PR[91] R[100]mm/sec CNT100;
   1:  PR[GP1:91,1] = PR[GP1:90,1] + 27.916;
   1:  PR[GP1:91,2] = PR[GP1:90,2] + 0.493;
   1:L PR[91] R[100]mm/sec CNT100;
   1:  PR[GP1:91,1] = PR[GP1:90,1] + 27.400;
   1:  PR[GP1:91,2] = PR[GP1:90,2] + 5.443;
   1:L PR[91] R[100]mm/sec CNT100;
   1:  PR[GP1:91,1] = PR[GP1:90,1] + 25.972;
   1:  PR[GP1:91,2] = PR[GP1:90,2] + 9.933;
   1:L PR[91] R[100]mm/sec CNT100;
   1:  PR[GP1:91,1] = PR[GP1:90,1] + 25.649;
   1:  PR[GP1:91,2] = PR[GP1:90,2] + 10.718;
   1:L PR[91] R[100]mm/sec CNT100;
   1:  PR[GP1:91,1] = PR[GP1:90,1] + 23.310;
   1:  PR[GP1:91,2] = PR[GP1:90,2] + 14.903;
   1:L PR[91] R[100]mm/sec CNT100;
   1:  PR[GP1:91,1] = PR[GP1:90,1] + 22.797;
   1:  PR[GP1:91,2] = PR[GP1:90,2] + 15.585;
   1:L PR[91] R[100]mm/sec CNT100;
   1:  PR[GP1:91,1] = PR[GP1:90,1] + 19.361;
   1:  PR[GP1:91,2] = PR[GP1:90,2] + 19.497;
   1:L PR[91] R[100]mm/sec CNT100;
   1:  PR[GP1:91,1] = PR[GP1:90,1] + 18.698;
   1:  PR[GP1:91,2] = PR[GP1:90,2] + 20.021;
   1:L PR[91] R[100]mm/sec CNT100;
   1:  PR[GP1:91,1] = PR[GP1:90,1] + 13.909;
   1:  PR[GP1:91,2] = PR[GP1:90,2] + 23.413;
   1:L PR[91] R[100]mm/sec CNT100;
   1:  PR[GP1:91,1] = PR[GP1:90,1] + 13.172;
   1:  PR[GP1:91,2] = PR[GP1:90,2] + 23.740;
   1:L PR[91] R[100]mm/sec CNT100;
   1:  PR[GP1:91,1] = PR[GP1:90,1] + 7.667;
   1:  PR[GP1:91,2] = PR[GP1:90,2] + 25.873;
   1:L PR[91] R[100]mm/sec CNT100;
   1:  PR[GP1:91,1] = PR[GP1:90,1] + 6.903;
   1:  PR[GP1:91,2] = PR[GP1:90,2] + 26.000;
   1:L PR[91] R[100]mm/sec CNT100;
   1:  PR[GP1:91,1] = PR[GP1:90,1] + 0.998;
   1:  PR[GP1:91,2] = PR[GP1:90,2] + 26.732;
   1:L PR[91] R[100]mm/sec CNT100;
   1:  PR[GP1:91,1] = PR[GP1:90,1] + 0.128;
   1:  PR[GP1:91,2] = PR[GP1:90,2] + 26.667;
   1:L PR[91] R[100]mm/sec CNT100;
   1:  PR[91] = PR[90];
   1:  PR[GP1:91,1] = PR[GP1:90,1] + -0.580;
   1:  PR[GP1:91,2] = PR[GP1:90,2] + 26.870;
   1:  PR[GP1:91,3] = PR[GP1:90,3] + 72.895;
   1:L PR[91] R[100]mm/sec CNT100;
   1:  PR[GP1:91,1] = PR[GP1:90,1] + -6.759;
   1:  PR[GP1:91,2] = PR[GP1:90,2] + 26.104;
   1:L PR[91] R[100]mm/sec CNT100;
   1:  PR[GP1:91,1] = PR[GP1:90,1] + -7.269;
   1:  PR[GP1:91,2] = PR[GP1:90,2] + 26.019;
   1:L PR[91] R[100]mm/sec CNT100;
   1:  PR[GP1:91,1] = PR[GP1:90,1] + -13.036;
   1:  PR[GP1:91,2] = PR[GP1:90,2] + 23.785;
   1:L PR[91] R[100]mm/sec CNT100;
   1:  PR[GP1:91,1] = PR[GP1:90,1] + -13.530;
   1:  PR[GP1:91,2] = PR[GP1:90,2] + 23.565;
   1:L PR[91] R[100]mm/sec CNT100;
   1:  PR[GP1:91,1] = PR[GP1:90,1] + -18.556;
   1:  PR[GP1:91,2] = PR[GP1:90,2] + 20.006;
   1:L PR[91] R[100]mm/sec CNT100;
   1:  PR[GP1:91,1] = PR[GP1:90,1] + -19.008;
   1:  PR[GP1:91,2] = PR[GP1:90,2] + 19.648;
   1:L PR[91] R[100]mm/sec CNT100;
   1:  PR[GP1:91,1] = PR[GP1:90,1] + -22.393;
   1:  PR[GP1:91,2] = PR[GP1:90,2] + 15.855;
   1:L PR[91] R[100]mm/sec CNT100;
   1:  PR[GP1:91,1] = PR[GP1:90,1] + -22.743;
   1:  PR[GP1:91,2] = PR[GP1:90,2] + 15.390;
   1:L PR[91] R[100]mm/sec CNT100;
   1:  PR[GP1:91,1] = PR[GP1:90,1] + -25.202;
   1:  PR[GP1:91,2] = PR[GP1:90,2] + 11.174;
   1:L PR[91] R[100]mm/sec CNT100;
   1:  PR[GP1:91,1] = PR[GP1:90,1] + -25.417;
   1:  PR[GP1:91,2] = PR[GP1:90,2] + 10.651;
   1:L PR[91] R[100]mm/sec CNT100;
   1:  PR[GP1:91,1] = PR[GP1:90,1] + -27.080;
   1:  PR[GP1:91,2] = PR[GP1:90,2] + 5.720;
   1:L PR[91] R[100]mm/sec CNT100;
   1:  PR[GP1:91,1] = PR[GP1:90,1] + -27.150;
   1:  PR[GP1:91,2] = PR[GP1:90,2] + 5.177;
   1:L PR[91] R[100]mm/sec CNT100;
   1:  PR[GP1:91,1] = PR[GP1:90,1] + -27.757;
   1:  PR[GP1:91,2] = PR[GP1:90,2] + -0.298;
   1:L PR[91] R[100]mm/sec CNT100;
   1:  PR[GP1:91,1] = PR[GP1:90,1] + -27.688;
   1:  PR[GP1:91,2] = PR[GP1:90,2] + -0.828;
   1:L PR[91] R[100]mm/sec CNT100;
   1:  PR[GP1:91,1] = PR[GP1:90,1] + -27.144;
   1:  PR[GP1:91,2] = PR[GP1:90,2] + -6.045;
   1:L PR[91] R[100]mm/sec CNT100;
   1:  PR[GP1:91,1] = PR[GP1:90,1] + -25.638;
   1:  PR[GP1:91,2] = PR[GP1:90,2] + -10.779;
   1:L PR[91] R[100]mm/sec CNT100;
   1:  PR[GP1:91,1] = PR[GP1:90,1] + -25.424;
   1:  PR[GP1:91,2] = PR[GP1:90,2] + -11.300;
   1:L PR[91] R[100]mm/sec CNT100;
   1:  PR[GP1:91,1] = PR[GP1:90,1] + -22.961;
   1:  PR[GP1:91,2] = PR[GP1:90,2] + -15.707;
   1:L PR[91] R[100]mm/sec CNT100;
   1:  PR[GP1:91,1] = PR[GP1:90,1] + -22.617;
   1:  PR[GP1:91,2] = PR[GP1:90,2] + -16.163;
   1:L PR[91] R[100]mm/sec CNT100;
   1:  PR[GP1:91,1] = PR[GP1:90,1] + -19.001;
   1:  PR[GP1:91,2] = PR[GP1:90,2] + -20.279;
   1:L PR[91] R[100]mm/sec CNT100;
   1:  PR[GP1:91,1] = PR[GP1:90,1] + -15.998;
   1:  PR[GP1:91,2] = PR[GP1:90,2] + -22.675;
   1:L PR[91] R[100]mm/sec CNT100;
   1:  PR[GP1:91,1] = PR[GP1:90,1] + -13.368;
   1:  PR[GP1:91,2] = PR[GP1:90,2] + -24.275;
   1:L PR[91] R[100]mm/sec CNT100;
   1:  PR[GP1:91,1] = PR[GP1:90,1] + -12.875;
   1:  PR[GP1:91,2] = PR[GP1:90,2] + -24.494;
   1:L PR[91] R[100]mm/sec CNT100;
   1:  PR[GP1:91,1] = PR[GP1:90,1] + -7.086;
   1:  PR[GP1:91,2] = PR[GP1:90,2] + -26.682;
   1:L PR[91] R[100]mm/sec CNT100;
   1:  PR[GP1:91,1] = PR[GP1:90,1] + -6.664;
   1:  PR[GP1:91,2] = PR[GP1:90,2] + -26.752;
   1:L PR[91] R[100]mm/sec CNT100;
   1:  PR[GP1:91,1] = PR[GP1:90,1] + -0.457;
   1:  PR[GP1:91,2] = PR[GP1:90,2] + -27.484;
   1:L PR[91] R[100]mm/sec CNT100;
   1:  PR[GP1:91,1] = PR[GP1:90,1] + 0.038;
   1:  PR[GP1:91,2] = PR[GP1:90,2] + -27.445;
   1:L PR[91] R[100]mm/sec CNT100;
   1:  PR[GP1:91,1] = PR[GP1:90,1] + 0.649;
   1:  PR[GP1:91,2] = PR[GP1:90,2] + -27.488;
   1:L PR[91] R[100]mm/sec CNT100;
   1:  PR[GP1:91,1] = PR[GP1:90,1] + 3.875;
   1:  PR[GP1:91,2] = PR[GP1:90,2] + -27.295;
   1:L PR[91] R[100]mm/sec CNT100;
   1:  PR[GP1:91,1] = PR[GP1:90,1] + 4.370;
   1:  PR[GP1:91,2] = PR[GP1:90,2] + -27.213;
   1:L PR[91] R[100]mm/sec CNT100;
   1:  PR[GP1:91,1] = PR[GP1:90,1] + 7.476;
   1:  PR[GP1:91,2] = PR[GP1:90,2] + -26.626;
   1:L PR[91] R[100]mm/sec CNT100;
   1:  PR[GP1:91,1] = PR[GP1:90,1] + 13.223;
   1:  PR[GP1:91,2] = PR[GP1:90,2] + -24.392;
   1:L PR[91] R[100]mm/sec CNT100;
   1:  PR[GP1:91,1] = PR[GP1:90,1] + 13.678;
   1:  PR[GP1:91,2] = PR[GP1:90,2] + -24.190;
   1:L PR[91] R[100]mm/sec CNT100;
   1:  PR[GP1:91,1] = PR[GP1:90,1] + 18.712;
   1:  PR[GP1:91,2] = PR[GP1:90,2] + -20.631;
   1:L PR[91] R[100]mm/sec CNT100;
   1:  PR[GP1:91,1] = PR[GP1:90,1] + 19.165;
   1:  PR[GP1:91,2] = PR[GP1:90,2] + -20.273;
   1:L PR[91] R[100]mm/sec CNT100;
   1:  PR[GP1:91,1] = PR[GP1:90,1] + 22.549;
   1:  PR[GP1:91,2] = PR[GP1:90,2] + -16.479;
   1:L PR[91] R[100]mm/sec CNT100;
   1:  PR[GP1:91,1] = PR[GP1:90,1] + 22.900;
   1:  PR[GP1:91,2] = PR[GP1:90,2] + -16.014;
   1:L PR[91] R[100]mm/sec CNT100;
   1:  PR[GP1:91,1] = PR[GP1:90,1] + 25.359;
   1:  PR[GP1:91,2] = PR[GP1:90,2] + -11.797;
   1:L PR[91] R[100]mm/sec CNT100;
   1:  PR[GP1:91,1] = PR[GP1:90,1] + 25.574;
   1:  PR[GP1:91,2] = PR[GP1:90,2] + -11.274;
   1:L PR[91] R[100]mm/sec CNT100;
   1:  PR[GP1:91,1] = PR[GP1:90,1] + 27.236;
   1:  PR[GP1:91,2] = PR[GP1:90,2] + -6.344;
   1:L PR[91] R[100]mm/sec CNT100;
   1:  PR[GP1:91,1] = PR[GP1:90,1] + 27.307;
   1:  PR[GP1:91,2] = PR[GP1:90,2] + -5.800;
   1:L PR[91] R[100]mm/sec CNT100;
   1:  PR[GP1:91,1] = PR[GP1:90,1] + 27.914;
   1:  PR[GP1:91,2] = PR[GP1:90,2] + -0.326;
   1:L PR[91] R[100]mm/sec CNT100;
   1:  PR[GP1:91,1] = PR[GP1:90,1] + 27.845;
   1:  PR[GP1:91,2] = PR[GP1:90,2] + 0.204;
   1:L PR[91] R[100]mm/sec CNT100;
   1:  PR[GP1:91,1] = PR[GP1:90,1] + 27.301;
   1:  PR[GP1:91,2] = PR[GP1:90,2] + 5.420;
   1:L PR[91] R[100]mm/sec CNT100;
   1:  PR[GP1:91,1] = PR[GP1:90,1] + 25.796;
   1:  PR[GP1:91,2] = PR[GP1:90,2] + 10.154;
   1:L PR[91] R[100]mm/sec CNT100;
   1:  PR[GP1:91,1] = PR[GP1:90,1] + 25.582;
   1:  PR[GP1:91,2] = PR[GP1:90,2] + 10.673;
   1:L PR[91] R[100]mm/sec CNT100;
   1:  PR[GP1:91,1] = PR[GP1:90,1] + 23.119;
   1:  PR[GP1:91,2] = PR[GP1:90,2] + 15.081;
   1:L PR[91] R[100]mm/sec CNT100;
   1:  PR[GP1:91,1] = PR[GP1:90,1] + 22.776;
   1:  PR[GP1:91,2] = PR[GP1:90,2] + 15.538;
   1:L PR[91] R[100]mm/sec CNT100;
   1:  PR[GP1:91,1] = PR[GP1:90,1] + 19.162;
   1:  PR[GP1:91,2] = PR[GP1:90,2] + 19.651;
   1:L PR[91] R[100]mm/sec CNT100;
   1:  PR[GP1:91,1] = PR[GP1:90,1] + 18.714;
   1:  PR[GP1:91,2] = PR[GP1:90,2] + 20.005;
   1:L PR[91] R[100]mm/sec CNT100;
   1:  PR[GP1:91,1] = PR[GP1:90,1] + 13.687;
   1:  PR[GP1:91,2] = PR[GP1:90,2] + 23.565;
   1:L PR[91] R[100]mm/sec CNT100;
   1:  PR[GP1:91,1] = PR[GP1:90,1] + 13.192;
   1:  PR[GP1:91,2] = PR[GP1:90,2] + 23.784;
   1:L PR[91] R[100]mm/sec CNT100;
   1:  PR[GP1:91,1] = PR[GP1:90,1] + 7.425;
   1:  PR[GP1:91,2] = PR[GP1:90,2] + 26.019;
   1:L PR[91] R[100]mm/sec CNT100;
   1:  PR[GP1:91,1] = PR[GP1:90,1] + 6.915;
   1:  PR[GP1:91,2] = PR[GP1:90,2] + 26.105;
   1:L PR[91] R[100]mm/sec CNT100;
   1:  PR[GP1:91,1] = PR[GP1:90,1] + 0.740;
   1:  PR[GP1:91,2] = PR[GP1:90,2] + 26.869;
   1:L PR[91] R[100]mm/sec CNT100;
   1:  PR[GP1:91,1] = PR[GP1:90,1] + 0.116;
   1:  PR[GP1:91,2] = PR[GP1:90,2] + 26.823;
   1:L PR[91] R[100]mm/sec CNT100;
   1:  PR[91] = PR[90];
   1:  PR[GP1:91,1] = PR[GP1:90,1] + -0.327;
   1:  PR[GP1:91,2] = PR[GP1:90,2] + 27.007;
   1:  PR[GP1:91,3] = PR[GP1:90,3] + 73.505;
   1:L PR[91] R[100]mm/sec CNT100;
   1:  PR[GP1:91,1] = PR[GP1:90,1] + -6.771;
   1:  PR[GP1:91,2] = PR[GP1:90,2] + 26.208;
   1:L PR[91] R[100]mm/sec CNT100;
   1:  PR[GP1:91,1] = PR[GP1:90,1] + -7.028;
   1:  PR[GP1:91,2] = PR[GP1:90,2] + 26.166;
   1:L PR[91] R[100]mm/sec CNT100;
   1:  PR[GP1:91,1] = PR[GP1:90,1] + -13.057;
   1:  PR[GP1:91,2] = PR[GP1:90,2] + 23.829;
   1:L PR[91] R[100]mm/sec CNT100;
   1:  PR[GP1:91,1] = PR[GP1:90,1] + -13.308;
   1:  PR[GP1:91,2] = PR[GP1:90,2] + 23.718;
   1:L PR[91] R[100]mm/sec CNT100;
   1:  PR[GP1:91,1] = PR[GP1:90,1] + -18.572;
   1:  PR[GP1:91,2] = PR[GP1:90,2] + 19.990;
   1:L PR[91] R[100]mm/sec CNT100;
   1:  PR[GP1:91,1] = PR[GP1:90,1] + -18.809;
   1:  PR[GP1:91,2] = PR[GP1:90,2] + 19.802;
   1:L PR[91] R[100]mm/sec CNT100;
   1:  PR[GP1:91,1] = PR[GP1:90,1] + -22.360;
   1:  PR[GP1:91,2] = PR[GP1:90,2] + 15.823;
   1:L PR[91] R[100]mm/sec CNT100;
   1:  PR[GP1:91,1] = PR[GP1:90,1] + -22.540;
   1:  PR[GP1:91,2] = PR[GP1:90,2] + 15.584;
   1:L PR[91] R[100]mm/sec CNT100;
   1:  PR[GP1:91,1] = PR[GP1:90,1] + -25.124;
   1:  PR[GP1:91,2] = PR[GP1:90,2] + 11.154;
   1:L PR[91] R[100]mm/sec CNT100;
   1:  PR[GP1:91,1] = PR[GP1:90,1] + -25.229;
   1:  PR[GP1:91,2] = PR[GP1:90,2] + 10.898;
   1:L PR[91] R[100]mm/sec CNT100;
   1:  PR[GP1:91,1] = PR[GP1:90,1] + -26.973;
   1:  PR[GP1:91,2] = PR[GP1:90,2] + 5.725;
   1:L PR[91] R[100]mm/sec CNT100;
   1:  PR[GP1:91,1] = PR[GP1:90,1] + -27.651;
   1:  PR[GP1:91,2] = PR[GP1:90,2] + -0.316;
   1:L PR[91] R[100]mm/sec CNT100;
   1:  PR[GP1:91,1] = PR[GP1:90,1] + -27.046;
   1:  PR[GP1:91,2] = PR[GP1:90,2] + -6.020;
   1:L PR[91] R[100]mm/sec CNT100;
   1:  PR[GP1:91,1] = PR[GP1:90,1] + -25.462;
   1:  PR[GP1:91,2] = PR[GP1:90,2] + -11.001;
   1:L PR[91] R[100]mm/sec CNT100;
   1:  PR[GP1:91,1] = PR[GP1:90,1] + -25.357;
   1:  PR[GP1:91,2] = PR[GP1:90,2] + -11.255;
   1:L PR[91] R[100]mm/sec CNT100;
   1:  PR[GP1:91,1] = PR[GP1:90,1] + -22.770;
   1:  PR[GP1:91,2] = PR[GP1:90,2] + -15.885;
   1:L PR[91] R[100]mm/sec CNT100;
   1:  PR[GP1:91,1] = PR[GP1:90,1] + -22.596;
   1:  PR[GP1:91,2] = PR[GP1:90,2] + -16.115;
   1:L PR[91] R[100]mm/sec CNT100;
   1:  PR[GP1:91,1] = PR[GP1:90,1] + -18.802;
   1:  PR[GP1:91,2] = PR[GP1:90,2] + -20.433;
   1:L PR[91] R[100]mm/sec CNT100;
   1:  PR[GP1:91,1] = PR[GP1:90,1] + -15.895;
   1:  PR[GP1:91,2] = PR[GP1:90,2] + -22.754;
   1:L PR[91] R[100]mm/sec CNT100;
   1:  PR[GP1:91,1] = PR[GP1:90,1] + -13.138;
   1:  PR[GP1:91,2] = PR[GP1:90,2] + -24.432;
   1:L PR[91] R[100]mm/sec CNT100;
   1:  PR[GP1:91,1] = PR[GP1:90,1] + -12.889;
   1:  PR[GP1:91,2] = PR[GP1:90,2] + -24.542;
   1:L PR[91] R[100]mm/sec CNT100;
   1:  PR[GP1:91,1] = PR[GP1:90,1] + -6.837;
   1:  PR[GP1:91,2] = PR[GP1:90,2] + -26.830;
   1:L PR[91] R[100]mm/sec CNT100;
   1:  PR[GP1:91,1] = PR[GP1:90,1] + -6.673;
   1:  PR[GP1:91,2] = PR[GP1:90,2] + -26.857;
   1:L PR[91] R[100]mm/sec CNT100;
   1:  PR[GP1:91,1] = PR[GP1:90,1] + -0.195;
   1:  PR[GP1:91,2] = PR[GP1:90,2] + -27.621;
   1:L PR[91] R[100]mm/sec CNT100;
   1:  PR[GP1:91,1] = PR[GP1:90,1] + 0.050;
   1:  PR[GP1:91,2] = PR[GP1:90,2] + -27.602;
   1:L PR[91] R[100]mm/sec CNT100;
   1:  PR[GP1:91,1] = PR[GP1:90,1] + 0.386;
   1:  PR[GP1:91,2] = PR[GP1:90,2] + -27.625;
   1:L PR[91] R[100]mm/sec CNT100;
   1:  PR[GP1:91,1] = PR[GP1:90,1] + 3.742;
   1:  PR[GP1:91,2] = PR[GP1:90,2] + -27.424;
   1:L PR[91] R[100]mm/sec CNT100;
   1:  PR[GP1:91,1] = PR[GP1:90,1] + 7.240;
   1:  PR[GP1:91,2] = PR[GP1:90,2] + -26.770;
   1:L PR[91] R[100]mm/sec CNT100;
   1:  PR[GP1:91,1] = PR[GP1:90,1] + 13.246;
   1:  PR[GP1:91,2] = PR[GP1:90,2] + -24.435;
   1:L PR[91] R[100]mm/sec CNT100;
   1:  PR[GP1:91,1] = PR[GP1:90,1] + 13.456;
   1:  PR[GP1:91,2] = PR[GP1:90,2] + -24.342;
   1:L PR[91] R[100]mm/sec CNT100;
   1:  PR[GP1:91,1] = PR[GP1:90,1] + 18.728;
   1:  PR[GP1:91,2] = PR[GP1:90,2] + -20.614;
   1:L PR[91] R[100]mm/sec CNT100;
   1:  PR[GP1:91,1] = PR[GP1:90,1] + 18.966;
   1:  PR[GP1:91,2] = PR[GP1:90,2] + -20.426;
   1:L PR[91] R[100]mm/sec CNT100;
   1:  PR[GP1:91,1] = PR[GP1:90,1] + 22.517;
   1:  PR[GP1:91,2] = PR[GP1:90,2] + -16.446;
   1:L PR[91] R[100]mm/sec CNT100;
   1:  PR[GP1:91,1] = PR[GP1:90,1] + 22.698;
   1:  PR[GP1:91,2] = PR[GP1:90,2] + -16.207;
   1:L PR[91] R[100]mm/sec CNT100;
   1:  PR[GP1:91,1] = PR[GP1:90,1] + 25.282;
   1:  PR[GP1:91,2] = PR[GP1:90,2] + -11.776;
   1:L PR[91] R[100]mm/sec CNT100;
   1:  PR[GP1:91,1] = PR[GP1:90,1] + 25.387;
   1:  PR[GP1:91,2] = PR[GP1:90,2] + -11.521;
   1:L PR[91] R[100]mm/sec CNT100;
   1:  PR[GP1:91,1] = PR[GP1:90,1] + 27.130;
   1:  PR[GP1:91,2] = PR[GP1:90,2] + -6.349;
   1:L PR[91] R[100]mm/sec CNT100;
   1:  PR[GP1:91,1] = PR[GP1:90,1] + 27.807;
   1:  PR[GP1:91,2] = PR[GP1:90,2] + -0.308;
   1:L PR[91] R[100]mm/sec CNT100;
   1:  PR[GP1:91,1] = PR[GP1:90,1] + 27.203;
   1:  PR[GP1:91,2] = PR[GP1:90,2] + 5.396;
   1:L PR[91] R[100]mm/sec CNT100;
   1:  PR[GP1:91,1] = PR[GP1:90,1] + 25.619;
   1:  PR[GP1:91,2] = PR[GP1:90,2] + 10.375;
   1:L PR[91] R[100]mm/sec CNT100;
   1:  PR[GP1:91,1] = PR[GP1:90,1] + 25.515;
   1:  PR[GP1:91,2] = PR[GP1:90,2] + 10.629;
   1:L PR[91] R[100]mm/sec CNT100;
   1:  PR[GP1:91,1] = PR[GP1:90,1] + 22.928;
   1:  PR[GP1:91,2] = PR[GP1:90,2] + 15.259;
   1:L PR[91] R[100]mm/sec CNT100;
   1:  PR[GP1:91,1] = PR[GP1:90,1] + 22.754;
   1:  PR[GP1:91,2] = PR[GP1:90,2] + 15.490;
   1:L PR[91] R[100]mm/sec CNT100;
   1:  PR[GP1:91,1] = PR[GP1:90,1] + 18.963;
   1:  PR[GP1:91,2] = PR[GP1:90,2] + 19.805;
   1:L PR[91] R[100]mm/sec CNT100;
   1:  PR[GP1:91,1] = PR[GP1:90,1] + 18.729;
   1:  PR[GP1:91,2] = PR[GP1:90,2] + 19.990;
   1:L PR[91] R[100]mm/sec CNT100;
   1:  PR[GP1:91,1] = PR[GP1:90,1] + 13.465;
   1:  PR[GP1:91,2] = PR[GP1:90,2] + 23.718;
   1:L PR[91] R[100]mm/sec CNT100;
   1:  PR[GP1:91,1] = PR[GP1:90,1] + 13.213;
   1:  PR[GP1:91,2] = PR[GP1:90,2] + 23.829;
   1:L PR[91] R[100]mm/sec CNT100;
   1:  PR[GP1:91,1] = PR[GP1:90,1] + 7.183;
   1:  PR[GP1:91,2] = PR[GP1:90,2] + 26.166;
   1:L PR[91] R[100]mm/sec CNT100;
   1:  PR[GP1:91,1] = PR[GP1:90,1] + 6.926;
   1:  PR[GP1:91,2] = PR[GP1:90,2] + 26.209;
   1:L PR[91] R[100]mm/sec CNT100;
   1:  PR[GP1:91,1] = PR[GP1:90,1] + 0.477;
   1:  PR[GP1:91,2] = PR[GP1:90,2] + 27.007;
   1:L PR[91] R[100]mm/sec CNT100;
   1:  PR[GP1:91,1] = PR[GP1:90,1] + 0.051;
   1:  PR[GP1:91,2] = PR[GP1:90,2] + 26.979;
   1:L PR[91] R[100]mm/sec CNT100;
   1:  PR[91] = PR[90];
   1:  PR[GP1:91,1] = PR[GP1:90,1] + -0.063;
   1:  PR[GP1:91,2] = PR[GP1:90,2] + 27.145;
   1:  PR[GP1:91,3] = PR[GP1:90,3] + 74.115;
   1:L PR[91] R[100]mm/sec CNT100;
   1:  PR[GP1:91,1] = PR[GP1:90,1] + -6.813;
   1:  PR[GP1:91,2] = PR[GP1:90,2] + 26.301;
   1:L PR[91] R[100]mm/sec CNT100;
   1:  PR[GP1:91,1] = PR[GP1:90,1] + -13.114;
   1:  PR[GP1:91,2] = PR[GP1:90,2] + 23.850;
   1:L PR[91] R[100]mm/sec CNT100;
   1:  PR[GP1:91,1] = PR[GP1:90,1] + -18.587;
   1:  PR[GP1:91,2] = PR[GP1:90,2] + 19.975;
   1:L PR[91] R[100]mm/sec CNT100;
   1:  PR[GP1:91,1] = PR[GP1:90,1] + -18.610;
   1:  PR[GP1:91,2] = PR[GP1:90,2] + 19.956;
   1:L PR[91] R[100]mm/sec CNT100;
   1:  PR[GP1:91,1] = PR[GP1:90,1] + -22.328;
   1:  PR[GP1:91,2] = PR[GP1:90,2] + 15.790;
   1:L PR[91] R[100]mm/sec CNT100;
   1:  PR[GP1:91,1] = PR[GP1:90,1] + -22.338;
   1:  PR[GP1:91,2] = PR[GP1:90,2] + 15.777;
   1:L PR[91] R[100]mm/sec CNT100;
   1:  PR[GP1:91,1] = PR[GP1:90,1] + -25.044;
   1:  PR[GP1:91,2] = PR[GP1:90,2] + 11.137;
   1:L PR[91] R[100]mm/sec CNT100;
   1:  PR[GP1:91,1] = PR[GP1:90,1] + -26.871;
   1:  PR[GP1:91,2] = PR[GP1:90,2] + 5.719;
   1:L PR[91] R[100]mm/sec CNT100;
   1:  PR[GP1:91,1] = PR[GP1:90,1] + -27.542;
   1:  PR[GP1:91,2] = PR[GP1:90,2] + -0.317;
   1:L PR[91] R[100]mm/sec CNT100;
   1:  PR[GP1:91,1] = PR[GP1:90,1] + -26.947;
   1:  PR[GP1:91,2] = PR[GP1:90,2] + -5.998;
   1:L PR[91] R[100]mm/sec CNT100;
   1:  PR[GP1:91,1] = PR[GP1:90,1] + -25.288;
   1:  PR[GP1:91,2] = PR[GP1:90,2] + -11.214;
   1:L PR[91] R[100]mm/sec CNT100;
   1:  PR[GP1:91,1] = PR[GP1:90,1] + -22.579;
   1:  PR[GP1:91,2] = PR[GP1:90,2] + -16.062;
   1:L PR[91] R[100]mm/sec CNT100;
   1:  PR[GP1:91,1] = PR[GP1:90,1] + -22.575;
   1:  PR[GP1:91,2] = PR[GP1:90,2] + -16.067;
   1:L PR[91] R[100]mm/sec CNT100;
   1:  PR[GP1:91,1] = PR[GP1:90,1] + -18.604;
   1:  PR[GP1:91,2] = PR[GP1:90,2] + -20.586;
   1:L PR[91] R[100]mm/sec CNT100;
   1:  PR[GP1:91,1] = PR[GP1:90,1] + -15.792;
   1:  PR[GP1:91,2] = PR[GP1:90,2] + -22.833;
   1:L PR[91] R[100]mm/sec CNT100;
   1:  PR[GP1:91,1] = PR[GP1:90,1] + -12.941;
   1:  PR[GP1:91,2] = PR[GP1:90,2] + -24.569;
   1:L PR[91] R[100]mm/sec CNT100;
   1:  PR[GP1:91,1] = PR[GP1:90,1] + -6.619;
   1:  PR[GP1:91,2] = PR[GP1:90,2] + -26.966;
   1:L PR[91] R[100]mm/sec CNT100;
   1:  PR[GP1:91,1] = PR[GP1:90,1] + 0.081;
   1:  PR[GP1:91,2] = PR[GP1:90,2] + -27.760;
   1:L PR[91] R[100]mm/sec CNT100;
   1:  PR[GP1:91,1] = PR[GP1:90,1] + 3.624;
   1:  PR[GP1:91,2] = PR[GP1:90,2] + -27.553;
   1:L PR[91] R[100]mm/sec CNT100;
   1:  PR[GP1:91,1] = PR[GP1:90,1] + 7.000;
   1:  PR[GP1:91,2] = PR[GP1:90,2] + -26.916;
   1:L PR[91] R[100]mm/sec CNT100;
   1:  PR[GP1:91,1] = PR[GP1:90,1] + 13.261;
   1:  PR[GP1:91,2] = PR[GP1:90,2] + -24.476;
   1:L PR[91] R[100]mm/sec CNT100;
   1:  PR[GP1:91,1] = PR[GP1:90,1] + 18.745;
   1:  PR[GP1:91,2] = PR[GP1:90,2] + -20.598;
   1:L PR[91] R[100]mm/sec CNT100;
   1:  PR[GP1:91,1] = PR[GP1:90,1] + 18.768;
   1:  PR[GP1:91,2] = PR[GP1:90,2] + -20.580;
   1:L PR[91] R[100]mm/sec CNT100;
   1:  PR[GP1:91,1] = PR[GP1:90,1] + 22.486;
   1:  PR[GP1:91,2] = PR[GP1:90,2] + -16.413;
   1:L PR[91] R[100]mm/sec CNT100;
   1:  PR[GP1:91,1] = PR[GP1:90,1] + 22.496;
   1:  PR[GP1:91,2] = PR[GP1:90,2] + -16.400;
   1:L PR[91] R[100]mm/sec CNT100;
   1:  PR[GP1:91,1] = PR[GP1:90,1] + 25.180;
   1:  PR[GP1:91,2] = PR[GP1:90,2] + -11.796;
   1:L PR[91] R[100]mm/sec CNT100;
   1:  PR[GP1:91,1] = PR[GP1:90,1] + 27.028;
   1:  PR[GP1:91,2] = PR[GP1:90,2] + -6.342;
   1:L PR[91] R[100]mm/sec CNT100;
   1:  PR[GP1:91,1] = PR[GP1:90,1] + 27.699;
   1:  PR[GP1:91,2] = PR[GP1:90,2] + -0.307;
   1:L PR[91] R[100]mm/sec CNT100;
   1:  PR[GP1:91,1] = PR[GP1:90,1] + 27.104;
   1:  PR[GP1:91,2] = PR[GP1:90,2] + 5.373;
   1:L PR[91] R[100]mm/sec CNT100;
   1:  PR[GP1:91,1] = PR[GP1:90,1] + 25.446;
   1:  PR[GP1:91,2] = PR[GP1:90,2] + 10.589;
   1:L PR[91] R[100]mm/sec CNT100;
   1:  PR[GP1:91,1] = PR[GP1:90,1] + 22.736;
   1:  PR[GP1:91,2] = PR[GP1:90,2] + 15.437;
   1:L PR[91] R[100]mm/sec CNT100;
   1:  PR[GP1:91,1] = PR[GP1:90,1] + 22.733;
   1:  PR[GP1:91,2] = PR[GP1:90,2] + 15.442;
   1:L PR[91] R[100]mm/sec CNT100;
   1:  PR[GP1:91,1] = PR[GP1:90,1] + 18.764;
   1:  PR[GP1:91,2] = PR[GP1:90,2] + 19.959;
   1:L PR[91] R[100]mm/sec CNT100;
   1:  PR[GP1:91,1] = PR[GP1:90,1] + 18.745;
   1:  PR[GP1:91,2] = PR[GP1:90,2] + 19.974;
   1:L PR[91] R[100]mm/sec CNT100;
   1:  PR[GP1:91,1] = PR[GP1:90,1] + 13.271;
   1:  PR[GP1:91,2] = PR[GP1:90,2] + 23.850;
   1:L PR[91] R[100]mm/sec CNT100;
   1:  PR[GP1:91,1] = PR[GP1:90,1] + 6.968;
   1:  PR[GP1:91,2] = PR[GP1:90,2] + 26.302;
   1:L PR[91] R[100]mm/sec CNT100;
   1:  PR[GP1:91,1] = PR[GP1:90,1] + 0.223;
   1:  PR[GP1:91,2] = PR[GP1:90,2] + 27.144;
   1:L PR[91] R[100]mm/sec CNT100;
   1:  PR[GP1:91,1] = PR[GP1:90,1] + 0.091;
   1:  PR[GP1:91,2] = PR[GP1:90,2] + 27.135;
   1:L PR[91] R[100]mm/sec CNT100;
   1:  PR[91] = PR[90];
   1:  PR[GP1:91,1] = PR[GP1:90,1] + -6.595;
   1:  PR[GP1:91,2] = PR[GP1:90,2] + 26.410;
   1:  PR[GP1:91,3] = PR[GP1:90,3] + 74.725;
   1:L PR[91] R[100]mm/sec CNT100;
   1:  PR[GP1:91,1] = PR[GP1:90,1] + -6.652;
   1:  PR[GP1:91,2] = PR[GP1:90,2] + 26.403;
   1:L PR[91] R[100]mm/sec CNT100;
   1:  PR[GP1:91,1] = PR[GP1:90,1] + -12.981;
   1:  PR[GP1:91,2] = PR[GP1:90,2] + 23.945;
   1:L PR[91] R[100]mm/sec CNT100;
   1:  PR[GP1:91,1] = PR[GP1:90,1] + -18.525;
   1:  PR[GP1:91,2] = PR[GP1:90,2] + 20.008;
   1:L PR[91] R[100]mm/sec CNT100;
   1:  PR[GP1:91,1] = PR[GP1:90,1] + -22.275;
   1:  PR[GP1:91,2] = PR[GP1:90,2] + 15.792;
   1:L PR[91] R[100]mm/sec CNT100;
   1:  PR[GP1:91,1] = PR[GP1:90,1] + -24.964;
   1:  PR[GP1:91,2] = PR[GP1:90,2] + 11.176;
   1:L PR[91] R[100]mm/sec CNT100;
   1:  PR[GP1:91,1] = PR[GP1:90,1] + -26.807;
   1:  PR[GP1:91,2] = PR[GP1:90,2] + 5.713;
   1:L PR[91] R[100]mm/sec CNT100;
   1:  PR[GP1:91,1] = PR[GP1:90,1] + -27.474;
   1:  PR[GP1:91,2] = PR[GP1:90,2] + -0.317;
   1:L PR[91] R[100]mm/sec CNT100;
   1:  PR[GP1:91,1] = PR[GP1:90,1] + -26.886;
   1:  PR[GP1:91,2] = PR[GP1:90,2] + -5.979;
   1:L PR[91] R[100]mm/sec CNT100;
   1:  PR[GP1:91,1] = PR[GP1:90,1] + -25.212;
   1:  PR[GP1:91,2] = PR[GP1:90,2] + -11.244;
   1:L PR[91] R[100]mm/sec CNT100;
   1:  PR[GP1:91,1] = PR[GP1:90,1] + -22.513;
   1:  PR[GP1:91,2] = PR[GP1:90,2] + -16.080;
   1:L PR[91] R[100]mm/sec CNT100;
   1:  PR[GP1:91,1] = PR[GP1:90,1] + -18.493;
   1:  PR[GP1:91,2] = PR[GP1:90,2] + -20.666;
   1:L PR[91] R[100]mm/sec CNT100;
   1:  PR[GP1:91,1] = PR[GP1:90,1] + -15.687;
   1:  PR[GP1:91,2] = PR[GP1:90,2] + -22.911;
   1:L PR[91] R[100]mm/sec CNT100;
   1:  PR[GP1:91,1] = PR[GP1:90,1] + -12.829;
   1:  PR[GP1:91,2] = PR[GP1:90,2] + -24.657;
   1:L PR[91] R[100]mm/sec CNT100;
   1:  PR[GP1:91,1] = PR[GP1:90,1] + -6.555;
   1:  PR[GP1:91,2] = PR[GP1:90,2] + -27.045;
   1:L PR[91] R[100]mm/sec CNT100;
   1:  PR[GP1:91,1] = PR[GP1:90,1] + 0.103;
   1:  PR[GP1:91,2] = PR[GP1:90,2] + -27.855;
   1:L PR[91] R[100]mm/sec CNT100;
   1:  PR[GP1:91,1] = PR[GP1:90,1] + 3.608;
   1:  PR[GP1:91,2] = PR[GP1:90,2] + -27.630;
   1:L PR[91] R[100]mm/sec CNT100;
   1:  PR[GP1:91,1] = PR[GP1:90,1] + 6.938;
   1:  PR[GP1:91,2] = PR[GP1:90,2] + -26.994;
   1:L PR[91] R[100]mm/sec CNT100;
   1:  PR[GP1:91,1] = PR[GP1:90,1] + 13.160;
   1:  PR[GP1:91,2] = PR[GP1:90,2] + -24.557;
   1:L PR[91] R[100]mm/sec CNT100;
   1:  PR[GP1:91,1] = PR[GP1:90,1] + 18.682;
   1:  PR[GP1:91,2] = PR[GP1:90,2] + -20.632;
   1:L PR[91] R[100]mm/sec CNT100;
   1:  PR[GP1:91,1] = PR[GP1:90,1] + 22.432;
   1:  PR[GP1:91,2] = PR[GP1:90,2] + -16.415;
   1:L PR[91] R[100]mm/sec CNT100;
   1:  PR[GP1:91,1] = PR[GP1:90,1] + 25.122;
   1:  PR[GP1:91,2] = PR[GP1:90,2] + -11.798;
   1:L PR[91] R[100]mm/sec CNT100;
   1:  PR[GP1:91,1] = PR[GP1:90,1] + 26.964;
   1:  PR[GP1:91,2] = PR[GP1:90,2] + -6.337;
   1:L PR[91] R[100]mm/sec CNT100;
   1:  PR[GP1:91,1] = PR[GP1:90,1] + 27.631;
   1:  PR[GP1:91,2] = PR[GP1:90,2] + -0.307;
   1:L PR[91] R[100]mm/sec CNT100;
   1:  PR[GP1:91,1] = PR[GP1:90,1] + 27.041;
   1:  PR[GP1:91,2] = PR[GP1:90,2] + 5.361;
   1:L PR[91] R[100]mm/sec CNT100;
   1:  PR[GP1:91,1] = PR[GP1:90,1] + 25.366;
   1:  PR[GP1:91,2] = PR[GP1:90,2] + 10.627;
   1:L PR[91] R[100]mm/sec CNT100;
   1:  PR[GP1:91,1] = PR[GP1:90,1] + 22.671;
   1:  PR[GP1:91,2] = PR[GP1:90,2] + 15.454;
   1:L PR[91] R[100]mm/sec CNT100;
   1:  PR[GP1:91,1] = PR[GP1:90,1] + 18.678;
   1:  PR[GP1:91,2] = PR[GP1:90,2] + 20.011;
   1:L PR[91] R[100]mm/sec CNT100;
   1:  PR[GP1:91,1] = PR[GP1:90,1] + 13.138;
   1:  PR[GP1:91,2] = PR[GP1:90,2] + 23.945;
   1:L PR[91] R[100]mm/sec CNT100;
   1:  PR[GP1:91,1] = PR[GP1:90,1] + 6.812;
   1:  PR[GP1:91,2] = PR[GP1:90,2] + 26.401;
   1:L PR[91] R[100]mm/sec CNT100;
   1:  PR[GP1:91,1] = PR[GP1:90,1] + 0.077;
   1:  PR[GP1:91,2] = PR[GP1:90,2] + 27.237;
   1:L PR[91] R[100]mm/sec CNT100;
   1:  PR[91] = PR[90];
   1:  PR[GP1:91,1] = PR[GP1:90,1] + -5.851;
   1:  PR[GP1:91,2] = PR[GP1:90,2] + 26.502;
   1:  PR[GP1:91,3] = PR[GP1:90,3] + 75.335;
   1:L PR[91] R[100]mm/sec CNT100;
   1:  PR[GP1:91,1] = PR[GP1:90,1] + -6.697;
   1:  PR[GP1:91,2] = PR[GP1:90,2] + 26.391;
   1:L PR[91] R[100]mm/sec CNT100;
   1:  PR[GP1:91,1] = PR[GP1:90,1] + -12.262;
   1:  PR[GP1:91,2] = PR[GP1:90,2] + 24.234;
   1:L PR[91] R[100]mm/sec CNT100;
   1:  PR[GP1:91,1] = PR[GP1:90,1] + -13.050;
   1:  PR[GP1:91,2] = PR[GP1:90,2] + 23.908;
   1:L PR[91] R[100]mm/sec CNT100;
   1:  PR[GP1:91,1] = PR[GP1:90,1] + -17.920;
   1:  PR[GP1:91,2] = PR[GP1:90,2] + 20.460;
   1:L PR[91] R[100]mm/sec CNT100;
   1:  PR[GP1:91,1] = PR[GP1:90,1] + -18.610;
   1:  PR[GP1:91,2] = PR[GP1:90,2] + 19.930;
   1:L PR[91] R[100]mm/sec CNT100;
   1:  PR[GP1:91,1] = PR[GP1:90,1] + -21.939;
   1:  PR[GP1:91,2] = PR[GP1:90,2] + 16.199;
   1:L PR[91] R[100]mm/sec CNT100;
   1:  PR[GP1:91,1] = PR[GP1:90,1] + -22.421;
   1:  PR[GP1:91,2] = PR[GP1:90,2] + 15.571;
   1:L PR[91] R[100]mm/sec CNT100;
   1:  PR[GP1:91,1] = PR[GP1:90,1] + -24.854;
   1:  PR[GP1:91,2] = PR[GP1:90,2] + 11.396;
   1:L PR[91] R[100]mm/sec CNT100;
   1:  PR[GP1:91,1] = PR[GP1:90,1] + -25.128;
   1:  PR[GP1:91,2] = PR[GP1:90,2] + 10.734;
   1:L PR[91] R[100]mm/sec CNT100;
   1:  PR[GP1:91,1] = PR[GP1:90,1] + -26.775;
   1:  PR[GP1:91,2] = PR[GP1:90,2] + 5.839;
   1:L PR[91] R[100]mm/sec CNT100;
   1:  PR[GP1:91,1] = PR[GP1:90,1] + -27.388;
   1:  PR[GP1:91,2] = PR[GP1:90,2] + 0.301;
   1:L PR[91] R[100]mm/sec CNT100;
   1:  PR[GP1:91,1] = PR[GP1:90,1] + -27.472;
   1:  PR[GP1:91,2] = PR[GP1:90,2] + -0.332;
   1:L PR[91] R[100]mm/sec CNT100;
   1:  PR[GP1:91,1] = PR[GP1:90,1] + -26.938;
   1:  PR[GP1:91,2] = PR[GP1:90,2] + -5.469;
   1:L PR[91] R[100]mm/sec CNT100;
   1:  PR[GP1:91,1] = PR[GP1:90,1] + -26.851;
   1:  PR[GP1:91,2] = PR[GP1:90,2] + -6.126;
   1:L PR[91] R[100]mm/sec CNT100;
   1:  PR[GP1:91,1] = PR[GP1:90,1] + -25.350;
   1:  PR[GP1:91,2] = PR[GP1:90,2] + -10.858;
   1:L PR[91] R[100]mm/sec CNT100;
   1:  PR[GP1:91,1] = PR[GP1:90,1] + -25.079;
   1:  PR[GP1:91,2] = PR[GP1:90,2] + -11.515;
   1:L PR[91] R[100]mm/sec CNT100;
   1:  PR[GP1:91,1] = PR[GP1:90,1] + -22.636;
   1:  PR[GP1:91,2] = PR[GP1:90,2] + -15.893;
   1:L PR[91] R[100]mm/sec CNT100;
   1:  PR[GP1:91,1] = PR[GP1:90,1] + -22.163;
   1:  PR[GP1:91,2] = PR[GP1:90,2] + -16.509;
   1:L PR[91] R[100]mm/sec CNT100;
   1:  PR[GP1:91,1] = PR[GP1:90,1] + -18.595;
   1:  PR[GP1:91,2] = PR[GP1:90,2] + -20.569;
   1:L PR[91] R[100]mm/sec CNT100;
   1:  PR[GP1:91,1] = PR[GP1:90,1] + -16.164;
   1:  PR[GP1:91,2] = PR[GP1:90,2] + -22.517;
   1:L PR[91] R[100]mm/sec CNT100;
   1:  PR[GP1:91,1] = PR[GP1:90,1] + -15.472;
   1:  PR[GP1:91,2] = PR[GP1:90,2] + -23.049;
   1:L PR[91] R[100]mm/sec CNT100;
   1:  PR[GP1:91,1] = PR[GP1:90,1] + -12.925;
   1:  PR[GP1:91,2] = PR[GP1:90,2] + -24.605;
   1:L PR[91] R[100]mm/sec CNT100;
   1:  PR[GP1:91,1] = PR[GP1:90,1] + -12.222;
   1:  PR[GP1:91,2] = PR[GP1:90,2] + -24.896;
   1:L PR[91] R[100]mm/sec CNT100;
   1:  PR[GP1:91,1] = PR[GP1:90,1] + -6.608;
   1:  PR[GP1:91,2] = PR[GP1:90,2] + -27.037;
   1:L PR[91] R[100]mm/sec CNT100;
   1:  PR[GP1:91,1] = PR[GP1:90,1] + 0.139;
   1:  PR[GP1:91,2] = PR[GP1:90,2] + -27.866;
   1:L PR[91] R[100]mm/sec CNT100;
   1:  PR[GP1:91,1] = PR[GP1:90,1] + 3.278;
   1:  PR[GP1:91,2] = PR[GP1:90,2] + -27.663;
   1:L PR[91] R[100]mm/sec CNT100;
   1:  PR[GP1:91,1] = PR[GP1:90,1] + 6.388;
   1:  PR[GP1:91,2] = PR[GP1:90,2] + -27.058;
   1:L PR[91] R[100]mm/sec CNT100;
   1:  PR[GP1:91,1] = PR[GP1:90,1] + 7.003;
   1:  PR[GP1:91,2] = PR[GP1:90,2] + -26.977;
   1:L PR[91] R[100]mm/sec CNT100;
   1:  PR[GP1:91,1] = PR[GP1:90,1] + 12.562;
   1:  PR[GP1:91,2] = PR[GP1:90,2] + -24.797;
   1:L PR[91] R[100]mm/sec CNT100;
   1:  PR[GP1:91,1] = PR[GP1:90,1] + 13.228;
   1:  PR[GP1:91,2] = PR[GP1:90,2] + -24.521;
   1:L PR[91] R[100]mm/sec CNT100;
   1:  PR[GP1:91,1] = PR[GP1:90,1] + 18.078;
   1:  PR[GP1:91,2] = PR[GP1:90,2] + -21.083;
   1:L PR[91] R[100]mm/sec CNT100;
   1:  PR[GP1:91,1] = PR[GP1:90,1] + 18.767;
   1:  PR[GP1:91,2] = PR[GP1:90,2] + -20.554;
   1:L PR[91] R[100]mm/sec CNT100;
   1:  PR[GP1:91,1] = PR[GP1:90,1] + 22.097;
   1:  PR[GP1:91,2] = PR[GP1:90,2] + -16.822;
   1:L PR[91] R[100]mm/sec CNT100;
   1:  PR[GP1:91,1] = PR[GP1:90,1] + 22.578;
   1:  PR[GP1:91,2] = PR[GP1:90,2] + -16.194;
   1:L PR[91] R[100]mm/sec CNT100;
   1:  PR[GP1:91,1] = PR[GP1:90,1] + 25.011;
   1:  PR[GP1:91,2] = PR[GP1:90,2] + -12.018;
   1:L PR[91] R[100]mm/sec CNT100;
   1:  PR[GP1:91,1] = PR[GP1:90,1] + 25.285;
   1:  PR[GP1:91,2] = PR[GP1:90,2] + -11.356;
   1:L PR[91] R[100]mm/sec CNT100;
   1:  PR[GP1:91,1] = PR[GP1:90,1] + 26.932;
   1:  PR[GP1:91,2] = PR[GP1:90,2] + -6.462;
   1:L PR[91] R[100]mm/sec CNT100;
   1:  PR[GP1:91,1] = PR[GP1:90,1] + 27.545;
   1:  PR[GP1:91,2] = PR[GP1:90,2] + -0.925;
   1:L PR[91] R[100]mm/sec CNT100;
   1:  PR[GP1:91,1] = PR[GP1:90,1] + 27.629;
   1:  PR[GP1:91,2] = PR[GP1:90,2] + -0.292;
   1:L PR[91] R[100]mm/sec CNT100;
   1:  PR[GP1:91,1] = PR[GP1:90,1] + 27.094;
   1:  PR[GP1:91,2] = PR[GP1:90,2] + 4.850;
   1:L PR[91] R[100]mm/sec CNT100;
   1:  PR[GP1:91,1] = PR[GP1:90,1] + 27.007;
   1:  PR[GP1:91,2] = PR[GP1:90,2] + 5.507;
   1:L PR[91] R[100]mm/sec CNT100;
   1:  PR[GP1:91,1] = PR[GP1:90,1] + 25.505;
   1:  PR[GP1:91,2] = PR[GP1:90,2] + 10.241;
   1:L PR[91] R[100]mm/sec CNT100;
   1:  PR[GP1:91,1] = PR[GP1:90,1] + 25.233;
   1:  PR[GP1:91,2] = PR[GP1:90,2] + 10.897;
   1:L PR[91] R[100]mm/sec CNT100;
   1:  PR[GP1:91,1] = PR[GP1:90,1] + 22.794;
   1:  PR[GP1:91,2] = PR[GP1:90,2] + 15.267;
   1:L PR[91] R[100]mm/sec CNT100;
   1:  PR[GP1:91,1] = PR[GP1:90,1] + 22.321;
   1:  PR[GP1:91,2] = PR[GP1:90,2] + 15.883;
   1:L PR[91] R[100]mm/sec CNT100;
   1:  PR[GP1:91,1] = PR[GP1:90,1] + 18.763;
   1:  PR[GP1:91,2] = PR[GP1:90,2] + 19.933;
   1:L PR[91] R[100]mm/sec CNT100;
   1:  PR[GP1:91,1] = PR[GP1:90,1] + 18.079;
   1:  PR[GP1:91,2] = PR[GP1:90,2] + 20.458;
   1:L PR[91] R[100]mm/sec CNT100;
   1:  PR[GP1:91,1] = PR[GP1:90,1] + 13.207;
   1:  PR[GP1:91,2] = PR[GP1:90,2] + 23.908;
   1:L PR[91] R[100]mm/sec CNT100;
   1:  PR[GP1:91,1] = PR[GP1:90,1] + 12.419;
   1:  PR[GP1:91,2] = PR[GP1:90,2] + 24.235;
   1:L PR[91] R[100]mm/sec CNT100;
   1:  PR[GP1:91,1] = PR[GP1:90,1] + 6.858;
   1:  PR[GP1:91,2] = PR[GP1:90,2] + 26.389;
   1:L PR[91] R[100]mm/sec CNT100;
   1:  PR[GP1:91,1] = PR[GP1:90,1] + 0.077;
   1:  PR[GP1:91,2] = PR[GP1:90,2] + 27.237;
   1:L PR[91] R[100]mm/sec CNT100;
   1:  PR[91] = PR[90];
   1:  PR[GP1:91,1] = PR[GP1:90,1] + -5.107;
   1:  PR[GP1:91,2] = PR[GP1:90,2] + 26.595;
   1:  PR[GP1:91,3] = PR[GP1:90,3] + 75.945;
   1:L PR[91] R[100]mm/sec CNT100;
   1:  PR[GP1:91,1] = PR[GP1:90,1] + -6.743;
   1:  PR[GP1:91,2] = PR[GP1:90,2] + 26.379;
   1:L PR[91] R[100]mm/sec CNT100;
   1:  PR[GP1:91,1] = PR[GP1:90,1] + -11.608;
   1:  PR[GP1:91,2] = PR[GP1:90,2] + 24.494;
   1:L PR[91] R[100]mm/sec CNT100;
   1:  PR[GP1:91,1] = PR[GP1:90,1] + -13.131;
   1:  PR[GP1:91,2] = PR[GP1:90,2] + 23.863;
   1:L PR[91] R[100]mm/sec CNT100;
   1:  PR[GP1:91,1] = PR[GP1:90,1] + -17.390;
   1:  PR[GP1:91,2] = PR[GP1:90,2] + 20.847;
   1:L PR[91] R[100]mm/sec CNT100;
   1:  PR[GP1:91,1] = PR[GP1:90,1] + -18.711;
   1:  PR[GP1:91,2] = PR[GP1:90,2] + 19.834;
   1:L PR[91] R[100]mm/sec CNT100;
   1:  PR[GP1:91,1] = PR[GP1:90,1] + -21.620;
   1:  PR[GP1:91,2] = PR[GP1:90,2] + 16.574;
   1:L PR[91] R[100]mm/sec CNT100;
   1:  PR[GP1:91,1] = PR[GP1:90,1] + -22.593;
   1:  PR[GP1:91,2] = PR[GP1:90,2] + 15.305;
   1:L PR[91] R[100]mm/sec CNT100;
   1:  PR[GP1:91,1] = PR[GP1:90,1] + -24.718;
   1:  PR[GP1:91,2] = PR[GP1:90,2] + 11.657;
   1:L PR[91] R[100]mm/sec CNT100;
   1:  PR[GP1:91,1] = PR[GP1:90,1] + -25.305;
   1:  PR[GP1:91,2] = PR[GP1:90,2] + 10.241;
   1:L PR[91] R[100]mm/sec CNT100;
   1:  PR[GP1:91,1] = PR[GP1:90,1] + -26.744;
   1:  PR[GP1:91,2] = PR[GP1:90,2] + 5.966;
   1:L PR[91] R[100]mm/sec CNT100;
   1:  PR[GP1:91,1] = PR[GP1:90,1] + -27.281;
   1:  PR[GP1:91,2] = PR[GP1:90,2] + 1.119;
   1:L PR[91] R[100]mm/sec CNT100;
   1:  PR[GP1:91,1] = PR[GP1:90,1] + -27.472;
   1:  PR[GP1:91,2] = PR[GP1:90,2] + -0.332;
   1:L PR[91] R[100]mm/sec CNT100;
   1:  PR[GP1:91,1] = PR[GP1:90,1] + -27.005;
   1:  PR[GP1:91,2] = PR[GP1:90,2] + -4.820;
   1:L PR[91] R[100]mm/sec CNT100;
   1:  PR[GP1:91,1] = PR[GP1:90,1] + -26.811;
   1:  PR[GP1:91,2] = PR[GP1:90,2] + -6.294;
   1:L PR[91] R[100]mm/sec CNT100;
   1:  PR[GP1:91,1] = PR[GP1:90,1] + -25.500;
   1:  PR[GP1:91,2] = PR[GP1:90,2] + -10.428;
   1:L PR[91] R[100]mm/sec CNT100;
   1:  PR[GP1:91,1] = PR[GP1:90,1] + -24.915;
   1:  PR[GP1:91,2] = PR[GP1:90,2] + -11.839;
   1:L PR[91] R[100]mm/sec CNT100;
   1:  PR[GP1:91,1] = PR[GP1:90,1] + -22.781;
   1:  PR[GP1:91,2] = PR[GP1:90,2] + -15.664;
   1:L PR[91] R[100]mm/sec CNT100;
   1:  PR[GP1:91,1] = PR[GP1:90,1] + -21.816;
   1:  PR[GP1:91,2] = PR[GP1:90,2] + -16.922;
   1:L PR[91] R[100]mm/sec CNT100;
   1:  PR[GP1:91,1] = PR[GP1:90,1] + -18.697;
   1:  PR[GP1:91,2] = PR[GP1:90,2] + -20.472;
   1:L PR[91] R[100]mm/sec CNT100;
   1:  PR[GP1:91,1] = PR[GP1:90,1] + -16.575;
   1:  PR[GP1:91,2] = PR[GP1:90,2] + -22.172;
   1:L PR[91] R[100]mm/sec CNT100;
   1:  PR[GP1:91,1] = PR[GP1:90,1] + -15.244;
   1:  PR[GP1:91,2] = PR[GP1:90,2] + -23.193;
   1:L PR[91] R[100]mm/sec CNT100;
   1:  PR[GP1:91,1] = PR[GP1:90,1] + -13.027;
   1:  PR[GP1:91,2] = PR[GP1:90,2] + -24.548;
   1:L PR[91] R[100]mm/sec CNT100;
   1:  PR[GP1:91,1] = PR[GP1:90,1] + -11.574;
   1:  PR[GP1:91,2] = PR[GP1:90,2] + -25.150;
   1:L PR[91] R[100]mm/sec CNT100;
   1:  PR[GP1:91,1] = PR[GP1:90,1] + -6.666;
   1:  PR[GP1:91,2] = PR[GP1:90,2] + -27.022;
   1:L PR[91] R[100]mm/sec CNT100;
   1:  PR[GP1:91,1] = PR[GP1:90,1] + -1.155;
   1:  PR[GP1:91,2] = PR[GP1:90,2] + -27.695;
   1:L PR[91] R[100]mm/sec CNT100;
   1:  PR[GP1:91,1] = PR[GP1:90,1] + 0.143;
   1:  PR[GP1:91,2] = PR[GP1:90,2] + -27.866;
   1:L PR[91] R[100]mm/sec CNT100;
   1:  PR[GP1:91,1] = PR[GP1:90,1] + 2.866;
   1:  PR[GP1:91,2] = PR[GP1:90,2] + -27.690;
   1:L PR[91] R[100]mm/sec CNT100;
   1:  PR[GP1:91,1] = PR[GP1:90,1] + 5.592;
   1:  PR[GP1:91,2] = PR[GP1:90,2] + -27.159;
   1:L PR[91] R[100]mm/sec CNT100;
   1:  PR[GP1:91,1] = PR[GP1:90,1] + 7.030;
   1:  PR[GP1:91,2] = PR[GP1:90,2] + -26.970;
   1:L PR[91] R[100]mm/sec CNT100;
   1:  PR[GP1:91,1] = PR[GP1:90,1] + 11.890;
   1:  PR[GP1:91,2] = PR[GP1:90,2] + -25.064;
   1:L PR[91] R[100]mm/sec CNT100;
   1:  PR[GP1:91,1] = PR[GP1:90,1] + 13.307;
   1:  PR[GP1:91,2] = PR[GP1:90,2] + -24.477;
   1:L PR[91] R[100]mm/sec CNT100;
   1:  PR[GP1:91,1] = PR[GP1:90,1] + 17.547;
   1:  PR[GP1:91,2] = PR[GP1:90,2] + -21.471;
   1:L PR[91] R[100]mm/sec CNT100;
   1:  PR[GP1:91,1] = PR[GP1:90,1] + 18.868;
   1:  PR[GP1:91,2] = PR[GP1:90,2] + -20.457;
   1:L PR[91] R[100]mm/sec CNT100;
   1:  PR[GP1:91,1] = PR[GP1:90,1] + 21.778;
   1:  PR[GP1:91,2] = PR[GP1:90,2] + -17.197;
   1:L PR[91] R[100]mm/sec CNT100;
   1:  PR[GP1:91,1] = PR[GP1:90,1] + 22.751;
   1:  PR[GP1:91,2] = PR[GP1:90,2] + -15.928;
   1:L PR[91] R[100]mm/sec CNT100;
   1:  PR[GP1:91,1] = PR[GP1:90,1] + 24.876;
   1:  PR[GP1:91,2] = PR[GP1:90,2] + -12.280;
   1:L PR[91] R[100]mm/sec CNT100;
   1:  PR[GP1:91,1] = PR[GP1:90,1] + 25.462;
   1:  PR[GP1:91,2] = PR[GP1:90,2] + -10.864;
   1:L PR[91] R[100]mm/sec CNT100;
   1:  PR[GP1:91,1] = PR[GP1:90,1] + 26.901;
   1:  PR[GP1:91,2] = PR[GP1:90,2] + -6.590;
   1:L PR[91] R[100]mm/sec CNT100;
   1:  PR[GP1:91,1] = PR[GP1:90,1] + 27.437;
   1:  PR[GP1:91,2] = PR[GP1:90,2] + -1.743;
   1:L PR[91] R[100]mm/sec CNT100;
   1:  PR[GP1:91,1] = PR[GP1:90,1] + 27.629;
   1:  PR[GP1:91,2] = PR[GP1:90,2] + -0.292;
   1:L PR[91] R[100]mm/sec CNT100;
   1:  PR[GP1:91,1] = PR[GP1:90,1] + 27.161;
   1:  PR[GP1:91,2] = PR[GP1:90,2] + 4.201;
   1:L PR[91] R[100]mm/sec CNT100;
   1:  PR[GP1:91,1] = PR[GP1:90,1] + 26.967;
   1:  PR[GP1:91,2] = PR[GP1:90,2] + 5.674;
   1:L PR[91] R[100]mm/sec CNT100;
   1:  PR[GP1:91,1] = PR[GP1:90,1] + 25.654;
   1:  PR[GP1:91,2] = PR[GP1:90,2] + 9.810;
   1:L PR[91] R[100]mm/sec CNT100;
   1:  PR[GP1:91,1] = PR[GP1:90,1] + 25.070;
   1:  PR[GP1:91,2] = PR[GP1:90,2] + 11.221;
   1:L PR[91] R[100]mm/sec CNT100;
   1:  PR[GP1:91,1] = PR[GP1:90,1] + 22.939;
   1:  PR[GP1:91,2] = PR[GP1:90,2] + 15.039;
   1:L PR[91] R[100]mm/sec CNT100;
   1:  PR[GP1:91,1] = PR[GP1:90,1] + 21.974;
   1:  PR[GP1:91,2] = PR[GP1:90,2] + 16.297;
   1:L PR[91] R[100]mm/sec CNT100;
   1:  PR[GP1:91,1] = PR[GP1:90,1] + 18.864;
   1:  PR[GP1:91,2] = PR[GP1:90,2] + 19.836;
   1:L PR[91] R[100]mm/sec CNT100;
   1:  PR[GP1:91,1] = PR[GP1:90,1] + 17.548;
   1:  PR[GP1:91,2] = PR[GP1:90,2] + 20.846;
   1:L PR[91] R[100]mm/sec CNT100;
   1:  PR[GP1:91,1] = PR[GP1:90,1] + 13.288;
   1:  PR[GP1:91,2] = PR[GP1:90,2] + 23.863;
   1:L PR[91] R[100]mm/sec CNT100;
   1:  PR[GP1:91,1] = PR[GP1:90,1] + 11.765;
   1:  PR[GP1:91,2] = PR[GP1:90,2] + 24.494;
   1:L PR[91] R[100]mm/sec CNT100;
   1:  PR[GP1:91,1] = PR[GP1:90,1] + 6.899;
   1:  PR[GP1:91,2] = PR[GP1:90,2] + 26.379;
   1:L PR[91] R[100]mm/sec CNT100;
   1:  PR[GP1:91,1] = PR[GP1:90,1] + 5.263;
   1:  PR[GP1:91,2] = PR[GP1:90,2] + 26.595;
   1:L PR[91] R[100]mm/sec CNT100;
   1:  PR[GP1:91,1] = PR[GP1:90,1] + 0.078;
   1:  PR[GP1:91,2] = PR[GP1:90,2] + 27.237;
   1:L PR[91] R[100]mm/sec CNT100;
   1:  PR[91] = PR[90];
   1:  PR[GP1:91,1] = PR[GP1:90,1] + -4.362;
   1:  PR[GP1:91,2] = PR[GP1:90,2] + 26.687;
   1:  PR[GP1:91,3] = PR[GP1:90,3] + 76.555;
   1:L PR[91] R[100]mm/sec CNT100;
   1:  PR[GP1:91,1] = PR[GP1:90,1] + -6.788;
   1:  PR[GP1:91,2] = PR[GP1:90,2] + 26.367;
   1:L PR[91] R[100]mm/sec CNT100;
   1:  PR[GP1:91,1] = PR[GP1:90,1] + -10.954;
   1:  PR[GP1:91,2] = PR[GP1:90,2] + 24.753;
   1:L PR[91] R[100]mm/sec CNT100;
   1:  PR[GP1:91,1] = PR[GP1:90,1] + -13.213;
   1:  PR[GP1:91,2] = PR[GP1:90,2] + 23.817;
   1:L PR[91] R[100]mm/sec CNT100;
   1:  PR[GP1:91,1] = PR[GP1:90,1] + -16.860;
   1:  PR[GP1:91,2] = PR[GP1:90,2] + 21.235;
   1:L PR[91] R[100]mm/sec CNT100;
   1:  PR[GP1:91,1] = PR[GP1:90,1] + -18.813;
   1:  PR[GP1:91,2] = PR[GP1:90,2] + 19.737;
   1:L PR[91] R[100]mm/sec CNT100;
   1:  PR[GP1:91,1] = PR[GP1:90,1] + -21.301;
   1:  PR[GP1:91,2] = PR[GP1:90,2] + 16.948;
   1:L PR[91] R[100]mm/sec CNT100;
   1:  PR[GP1:91,1] = PR[GP1:90,1] + -22.766;
   1:  PR[GP1:91,2] = PR[GP1:90,2] + 15.038;
   1:L PR[91] R[100]mm/sec CNT100;
   1:  PR[GP1:91,1] = PR[GP1:90,1] + -24.583;
   1:  PR[GP1:91,2] = PR[GP1:90,2] + 11.919;
   1:L PR[91] R[100]mm/sec CNT100;
   1:  PR[GP1:91,1] = PR[GP1:90,1] + -25.482;
   1:  PR[GP1:91,2] = PR[GP1:90,2] + 9.749;
   1:L PR[91] R[100]mm/sec CNT100;
   1:  PR[GP1:91,1] = PR[GP1:90,1] + -26.713;
   1:  PR[GP1:91,2] = PR[GP1:90,2] + 6.093;
   1:L PR[91] R[100]mm/sec CNT100;
   1:  PR[GP1:91,1] = PR[GP1:90,1] + -27.173;
   1:  PR[GP1:91,2] = PR[GP1:90,2] + 1.937;
   1:L PR[91] R[100]mm/sec CNT100;
   1:  PR[GP1:91,1] = PR[GP1:90,1] + -27.472;
   1:  PR[GP1:91,2] = PR[GP1:90,2] + -0.332;
   1:L PR[91] R[100]mm/sec CNT100;
   1:  PR[GP1:91,1] = PR[GP1:90,1] + -27.073;
   1:  PR[GP1:91,2] = PR[GP1:90,2] + -4.172;
   1:L PR[91] R[100]mm/sec CNT100;
   1:  PR[GP1:91,1] = PR[GP1:90,1] + -26.771;
   1:  PR[GP1:91,2] = PR[GP1:90,2] + -6.462;
   1:L PR[91] R[100]mm/sec CNT100;
   1:  PR[GP1:91,1] = PR[GP1:90,1] + -25.650;
   1:  PR[GP1:91,2] = PR[GP1:90,2] + -9.998;
   1:L PR[91] R[100]mm/sec CNT100;
   1:  PR[GP1:91,1] = PR[GP1:90,1] + -24.752;
   1:  PR[GP1:91,2] = PR[GP1:90,2] + -12.164;
   1:L PR[91] R[100]mm/sec CNT100;
   1:  PR[GP1:91,1] = PR[GP1:90,1] + -22.927;
   1:  PR[GP1:91,2] = PR[GP1:90,2] + -15.436;
   1:L PR[91] R[100]mm/sec CNT100;
   1:  PR[GP1:91,1] = PR[GP1:90,1] + -21.469;
   1:  PR[GP1:91,2] = PR[GP1:90,2] + -17.336;
   1:L PR[91] R[100]mm/sec CNT100;
   1:  PR[GP1:91,1] = PR[GP1:90,1] + -18.798;
   1:  PR[GP1:91,2] = PR[GP1:90,2] + -20.375;
   1:L PR[91] R[100]mm/sec CNT100;
   1:  PR[GP1:91,1] = PR[GP1:90,1] + -16.986;
   1:  PR[GP1:91,2] = PR[GP1:90,2] + -21.827;
   1:L PR[91] R[100]mm/sec CNT100;
   1:  PR[GP1:91,1] = PR[GP1:90,1] + -15.017;
   1:  PR[GP1:91,2] = PR[GP1:90,2] + -23.338;
   1:L PR[91] R[100]mm/sec CNT100;
   1:  PR[GP1:91,1] = PR[GP1:90,1] + -13.129;
   1:  PR[GP1:91,2] = PR[GP1:90,2] + -24.491;
   1:L PR[91] R[100]mm/sec CNT100;
   1:  PR[GP1:91,1] = PR[GP1:90,1] + -10.925;
   1:  PR[GP1:91,2] = PR[GP1:90,2] + -25.404;
   1:L PR[91] R[100]mm/sec CNT100;
   1:  PR[GP1:91,1] = PR[GP1:90,1] + -6.723;
   1:  PR[GP1:91,2] = PR[GP1:90,2] + -27.007;
   1:L PR[91] R[100]mm/sec CNT100;
   1:  PR[GP1:91,1] = PR[GP1:90,1] + -2.000;
   1:  PR[GP1:91,2] = PR[GP1:90,2] + -27.584;
   1:L PR[91] R[100]mm/sec CNT100;
   1:  PR[GP1:91,1] = PR[GP1:90,1] + 0.140;
   1:  PR[GP1:91,2] = PR[GP1:90,2] + -27.866;
   1:L PR[91] R[100]mm/sec CNT100;
   1:  PR[GP1:91,1] = PR[GP1:90,1] + 2.454;
   1:  PR[GP1:91,2] = PR[GP1:90,2] + -27.716;
   1:L PR[91] R[100]mm/sec CNT100;
   1:  PR[GP1:91,1] = PR[GP1:90,1] + 4.795;
   1:  PR[GP1:91,2] = PR[GP1:90,2] + -27.260;
   1:L PR[91] R[100]mm/sec CNT100;
   1:  PR[GP1:91,1] = PR[GP1:90,1] + 7.057;
   1:  PR[GP1:91,2] = PR[GP1:90,2] + -26.962;
   1:L PR[91] R[100]mm/sec CNT100;
   1:  PR[GP1:91,1] = PR[GP1:90,1] + 11.219;
   1:  PR[GP1:91,2] = PR[GP1:90,2] + -25.330;
   1:L PR[91] R[100]mm/sec CNT100;
   1:  PR[GP1:91,1] = PR[GP1:90,1] + 13.386;
   1:  PR[GP1:91,2] = PR[GP1:90,2] + -24.433;
   1:L PR[91] R[100]mm/sec CNT100;
   1:  PR[GP1:91,1] = PR[GP1:90,1] + 17.017;
   1:  PR[GP1:91,2] = PR[GP1:90,2] + -21.858;
   1:L PR[91] R[100]mm/sec CNT100;
   1:  PR[GP1:91,1] = PR[GP1:90,1] + 18.970;
   1:  PR[GP1:91,2] = PR[GP1:90,2] + -20.360;
   1:L PR[91] R[100]mm/sec CNT100;
   1:  PR[GP1:91,1] = PR[GP1:90,1] + 21.458;
   1:  PR[GP1:91,2] = PR[GP1:90,2] + -17.571;
   1:L PR[91] R[100]mm/sec CNT100;
   1:  PR[GP1:91,1] = PR[GP1:90,1] + 22.923;
   1:  PR[GP1:91,2] = PR[GP1:90,2] + -15.662;
   1:L PR[91] R[100]mm/sec CNT100;
   1:  PR[GP1:91,1] = PR[GP1:90,1] + 24.741;
   1:  PR[GP1:91,2] = PR[GP1:90,2] + -12.542;
   1:L PR[91] R[100]mm/sec CNT100;
   1:  PR[GP1:91,1] = PR[GP1:90,1] + 25.640;
   1:  PR[GP1:91,2] = PR[GP1:90,2] + -10.372;
   1:L PR[91] R[100]mm/sec CNT100;
   1:  PR[GP1:91,1] = PR[GP1:90,1] + 26.870;
   1:  PR[GP1:91,2] = PR[GP1:90,2] + -6.717;
   1:L PR[91] R[100]mm/sec CNT100;
   1:  PR[GP1:91,1] = PR[GP1:90,1] + 27.330;
   1:  PR[GP1:91,2] = PR[GP1:90,2] + -2.561;
   1:L PR[91] R[100]mm/sec CNT100;
   1:  PR[GP1:91,1] = PR[GP1:90,1] + 27.629;
   1:  PR[GP1:91,2] = PR[GP1:90,2] + -0.292;
   1:L PR[91] R[100]mm/sec CNT100;
   1:  PR[GP1:91,1] = PR[GP1:90,1] + 27.229;
   1:  PR[GP1:91,2] = PR[GP1:90,2] + 3.552;
   1:L PR[91] R[100]mm/sec CNT100;
   1:  PR[GP1:91,1] = PR[GP1:90,1] + 26.927;
   1:  PR[GP1:91,2] = PR[GP1:90,2] + 5.841;
   1:L PR[91] R[100]mm/sec CNT100;
   1:  PR[GP1:91,1] = PR[GP1:90,1] + 25.804;
   1:  PR[GP1:91,2] = PR[GP1:90,2] + 9.379;
   1:L PR[91] R[100]mm/sec CNT100;
   1:  PR[GP1:91,1] = PR[GP1:90,1] + 24.907;
   1:  PR[GP1:91,2] = PR[GP1:90,2] + 11.545;
   1:L PR[91] R[100]mm/sec CNT100;
   1:  PR[GP1:91,1] = PR[GP1:90,1] + 23.084;
   1:  PR[GP1:91,2] = PR[GP1:90,2] + 14.811;
   1:L PR[91] R[100]mm/sec CNT100;
   1:  PR[GP1:91,1] = PR[GP1:90,1] + 21.627;
   1:  PR[GP1:91,2] = PR[GP1:90,2] + 16.711;
   1:L PR[91] R[100]mm/sec CNT100;
   1:  PR[GP1:91,1] = PR[GP1:90,1] + 18.966;
   1:  PR[GP1:91,2] = PR[GP1:90,2] + 19.740;
   1:L PR[91] R[100]mm/sec CNT100;
   1:  PR[GP1:91,1] = PR[GP1:90,1] + 17.018;
   1:  PR[GP1:91,2] = PR[GP1:90,2] + 21.234;
   1:L PR[91] R[100]mm/sec CNT100;
   1:  PR[GP1:91,1] = PR[GP1:90,1] + 13.370;
   1:  PR[GP1:91,2] = PR[GP1:90,2] + 23.817;
   1:L PR[91] R[100]mm/sec CNT100;
   1:  PR[GP1:91,1] = PR[GP1:90,1] + 11.111;
   1:  PR[GP1:91,2] = PR[GP1:90,2] + 24.753;
   1:L PR[91] R[100]mm/sec CNT100;
   1:  PR[GP1:91,1] = PR[GP1:90,1] + 6.944;
   1:  PR[GP1:91,2] = PR[GP1:90,2] + 26.368;
   1:L PR[91] R[100]mm/sec CNT100;
   1:  PR[GP1:91,1] = PR[GP1:90,1] + 4.519;
   1:  PR[GP1:91,2] = PR[GP1:90,2] + 26.687;
   1:L PR[91] R[100]mm/sec CNT100;
   1:  PR[GP1:91,1] = PR[GP1:90,1] + 0.078;
   1:  PR[GP1:91,2] = PR[GP1:90,2] + 27.237;
   1:L PR[91] R[100]mm/sec CNT100;
   1:  PR[91] = PR[90];
   1:  PR[GP1:91,1] = PR[GP1:90,1] + -3.618;
   1:  PR[GP1:91,2] = PR[GP1:90,2] + 26.779;
   1:  PR[GP1:91,3] = PR[GP1:90,3] + 77.165;
   1:L PR[91] R[100]mm/sec CNT100;
   1:  PR[GP1:91,1] = PR[GP1:90,1] + -6.833;
   1:  PR[GP1:91,2] = PR[GP1:90,2] + 26.356;
   1:L PR[91] R[100]mm/sec CNT100;
   1:  PR[GP1:91,1] = PR[GP1:90,1] + -10.301;
   1:  PR[GP1:91,2] = PR[GP1:90,2] + 25.012;
   1:L PR[91] R[100]mm/sec CNT100;
   1:  PR[GP1:91,1] = PR[GP1:90,1] + -13.295;
   1:  PR[GP1:91,2] = PR[GP1:90,2] + 23.772;
   1:L PR[91] R[100]mm/sec CNT100;
   1:  PR[GP1:91,1] = PR[GP1:90,1] + -16.330;
   1:  PR[GP1:91,2] = PR[GP1:90,2] + 21.623;
   1:L PR[91] R[100]mm/sec CNT100;
   1:  PR[GP1:91,1] = PR[GP1:90,1] + -18.914;
   1:  PR[GP1:91,2] = PR[GP1:90,2] + 19.640;
   1:L PR[91] R[100]mm/sec CNT100;
   1:  PR[GP1:91,1] = PR[GP1:90,1] + -20.982;
   1:  PR[GP1:91,2] = PR[GP1:90,2] + 17.323;
   1:L PR[91] R[100]mm/sec CNT100;
   1:  PR[GP1:91,1] = PR[GP1:90,1] + -22.939;
   1:  PR[GP1:91,2] = PR[GP1:90,2] + 14.772;
   1:L PR[91] R[100]mm/sec CNT100;
   1:  PR[GP1:91,1] = PR[GP1:90,1] + -24.448;
   1:  PR[GP1:91,2] = PR[GP1:90,2] + 12.181;
   1:L PR[91] R[100]mm/sec CNT100;
   1:  PR[GP1:91,1] = PR[GP1:90,1] + -25.660;
   1:  PR[GP1:91,2] = PR[GP1:90,2] + 9.256;
   1:L PR[91] R[100]mm/sec CNT100;
   1:  PR[GP1:91,1] = PR[GP1:90,1] + -26.682;
   1:  PR[GP1:91,2] = PR[GP1:90,2] + 6.220;
   1:L PR[91] R[100]mm/sec CNT100;
   1:  PR[GP1:91,1] = PR[GP1:90,1] + -27.065;
   1:  PR[GP1:91,2] = PR[GP1:90,2] + 2.756;
   1:L PR[91] R[100]mm/sec CNT100;
   1:  PR[GP1:91,1] = PR[GP1:90,1] + -27.472;
   1:  PR[GP1:91,2] = PR[GP1:90,2] + -0.332;
   1:L PR[91] R[100]mm/sec CNT100;
   1:  PR[GP1:91,1] = PR[GP1:90,1] + -27.140;
   1:  PR[GP1:91,2] = PR[GP1:90,2] + -3.524;
   1:L PR[91] R[100]mm/sec CNT100;
   1:  PR[GP1:91,1] = PR[GP1:90,1] + -26.731;
   1:  PR[GP1:91,2] = PR[GP1:90,2] + -6.629;
   1:L PR[91] R[100]mm/sec CNT100;
   1:  PR[GP1:91,1] = PR[GP1:90,1] + -25.799;
   1:  PR[GP1:91,2] = PR[GP1:90,2] + -9.568;
   1:L PR[91] R[100]mm/sec CNT100;
   1:  PR[GP1:91,1] = PR[GP1:90,1] + -24.589;
   1:  PR[GP1:91,2] = PR[GP1:90,2] + -12.489;
   1:L PR[91] R[100]mm/sec CNT100;
   1:  PR[GP1:91,1] = PR[GP1:90,1] + -23.072;
   1:  PR[GP1:91,2] = PR[GP1:90,2] + -15.208;
   1:L PR[91] R[100]mm/sec CNT100;
   1:  PR[GP1:91,1] = PR[GP1:90,1] + -21.122;
   1:  PR[GP1:91,2] = PR[GP1:90,2] + -17.749;
   1:L PR[91] R[100]mm/sec CNT100;
   1:  PR[GP1:91,1] = PR[GP1:90,1] + -18.900;
   1:  PR[GP1:91,2] = PR[GP1:90,2] + -20.279;
   1:L PR[91] R[100]mm/sec CNT100;
   1:  PR[GP1:91,1] = PR[GP1:90,1] + -17.397;
   1:  PR[GP1:91,2] = PR[GP1:90,2] + -21.483;
   1:L PR[91] R[100]mm/sec CNT100;
   1:  PR[GP1:91,1] = PR[GP1:90,1] + -14.790;
   1:  PR[GP1:91,2] = PR[GP1:90,2] + -23.483;
   1:L PR[91] R[100]mm/sec CNT100;
   1:  PR[GP1:91,1] = PR[GP1:90,1] + -13.232;
   1:  PR[GP1:91,2] = PR[GP1:90,2] + -24.435;
   1:L PR[91] R[100]mm/sec CNT100;
   1:  PR[GP1:91,1] = PR[GP1:90,1] + -10.277;
   1:  PR[GP1:91,2] = PR[GP1:90,2] + -25.659;
   1:L PR[91] R[100]mm/sec CNT100;
   1:  PR[GP1:91,1] = PR[GP1:90,1] + -6.780;
   1:  PR[GP1:91,2] = PR[GP1:90,2] + -26.992;
   1:L PR[91] R[100]mm/sec CNT100;
   1:  PR[GP1:91,1] = PR[GP1:90,1] + -2.844;
